LIN {X 0,Y 442.368,Z 762.06,A -85,B 0,C 180,E1 14751.098,E2 14751.098} C_VEL
LIN {X 0,Y 442.765,Z 762.06,A -85,B 0,C 180,E1 14758.998,E2 14758.998} C_VEL
LIN {X 0,Y 442.299,Z 762.06,A -85,B 0,C 180,E1 14768.863,E2 14768.863} C_VEL
LIN {X 0,Y 442.48,Z 764.15,A -85,B 0,C 180,E1 14772.989,E2 14772.989} C_VEL
LIN {X 0,Y 454.575,Z 779.497,A -85,B 0,C 180,E1 14779.866,E2 14779.866} C_VEL
LIN {X 0,Y 479.649,Z 812.394,A -85,B 0,C 180,E1 14788.603,E2 14788.603} C_VEL
LIN {X 0,Y 507.848,Z 858.532,A -85,B 0,C 180,E1 14795.89,E2 14795.89} C_VEL
LIN {X 0,Y 520.957,Z 891.034,A -85,B 0,C 180,E1 14799.521,E2 14799.521} C_VEL
LIN {X 0,Y 506.276,Z 963.742,A -85,B 0,C 180,E1 14802.79,E2 14802.79} C_VEL
LIN {X 0,Y 487.966,Z 1029.094,A -85,B 0,C 180,E1 14807.79,E2 14807.79} C_VEL
LIN {X 0,Y 469.666,Z 1084.518,A -85,B 0,C 180,E1 14814.467,E2 14814.467} C_VEL
LIN {X 0,Y 454.767,Z 1129.328,A -85,B 0,C 180,E1 14822.874,E2 14822.874} C_VEL
LIN {X 0,Y 446.413,Z 1161.096,A -85,B 0,C 180,E1 14832.529,E2 14832.529} C_VEL
LIN {X 0,Y 443.437,Z 1178.275,A -85,B 0,C 180,E1 14842.403,E2 14842.403} C_VEL
LIN {X 0,Y 443.471,Z 1182.026,A -85,B 0,C 180,E1 14850.982,E2 14850.982} C_VEL
LIN {X 0,Y 443.626,Z 1175.498,A -85,B 0,C 180,E1 14859.843,E2 14859.843} C_VEL
LIN {X 0,Y 447.223,Z 1156.157,A -85,B 0,C 180,E1 14869.308,E2 14869.308} C_VEL
LIN {X 0,Y 457.262,Z 1121.757,A -85,B 0,C 180,E1 14878.746,E2 14878.746} C_VEL
LIN {X 0,Y 473.14,Z 1074.147,A -85,B 0,C 180,E1 14886.926,E2 14886.926} C_VEL
LIN {X 0,Y 491.971,Z 1015.812,A -85,B 0,C 180,E1 14893.329,E2 14893.329} C_VEL
LIN {X 0,Y 509.871,Z 949.056,A -85,B 0,C 180,E1 14897.908,E2 14897.908} C_VEL
LIN {X 0,Y 520.404,Z 886.291,A -85,B 0,C 180,E1 14900.698,E2 14900.698} C_VEL
LIN {X 0,Y 494.713,Z 835.568,A -85,B 0,C 180,E1 14907.281,E2 14907.281} C_VEL
LIN {X 0,Y 467.97,Z 797.024,A -85,B 0,C 180,E1 14914.818,E2 14914.818} C_VEL
LIN {X 0,Y 451.114,Z 775.579,A -85,B 0,C 180,E1 14921.571,E2 14921.571} C_VEL
LIN {X 0,Y 445.46,Z 768.317,A -85,B 0,C 180,E1 14924.718,E2 14924.718} C_VEL
LIN {X 0,Y 442.777,Z 762.06,A -85,B 0,C 180,E1 14927.464,E2 14927.464} C_VEL
LIN {X 0,Y 442.754,Z 762.06,A -85,B 0,C 180,E1 14939.038,E2 14939.038} C_VEL
LIN {X 0,Y 442.287,Z 762.234,A -85,B 0,C 180,E1 14949.091,E2 14949.091} C_VEL
LIN {X 0,Y 459.966,Z 786.242,A -85,B 0,C 180,E1 14958.467,E2 14958.467} C_VEL
LIN {X 0,Y 486.214,Z 823.053,A -85,B 0,C 180,E1 14966.809,E2 14966.809} C_VEL
LIN {X 0,Y 512.137,Z 870.616,A -85,B 0,C 180,E1 14973.588,E2 14973.588} C_VEL
LIN {X 0,Y 521.201,Z 897.2,A -85,B 0,C 180,E1 14976.35,E2 14976.35} C_VEL
LIN {X 0,Y 506.051,Z 970.977,A -85,B 0,C 180,E1 14979.792,E2 14979.792} C_VEL
LIN {X 0,Y 487.203,Z 1040.281,A -85,B 0,C 180,E1 14985.118,E2 14985.118} C_VEL
LIN {X 0,Y 469.206,Z 1099.476,A -85,B 0,C 180,E1 14992.154,E2 14992.154} C_VEL
LIN {X 0,Y 454.918,Z 1147.637,A -85,B 0,C 180,E1 15000.758,E2 15000.758} C_VEL
LIN {X 0,Y 446.328,Z 1183.36,A -85,B 0,C 180,E1 15010.651,E2 15010.651} C_VEL
LIN {X 0,Y 443.387,Z 1202.811,A -85,B 0,C 180,E1 15020.151,E2 15020.151} C_VEL
LIN {X 0,Y 443.483,Z 1209.43,A -85,B 0,C 180,E1 15029.018,E2 15029.018} C_VEL
LIN {X 0,Y 443.218,Z 1205.935,A -85,B 0,C 180,E1 15037.185,E2 15037.185} C_VEL
LIN {X 0,Y 435.795,Z 1200.131,A -85,B 0,C 180,E1 15041.665,E2 15041.665} C_VEL
LIN {X 0,Y 439.135,Z 1178.691,A -85,B 0,C 180,E1 15051.258,E2 15051.258} C_VEL
LIN {X 0,Y 448.542,Z 1142.903,A -85,B 0,C 180,E1 15060.768,E2 15060.768} C_VEL
LIN {X 0,Y 464.675,Z 1092.053,A -85,B 0,C 180,E1 15069.522,E2 15069.522} C_VEL
LIN {X 0,Y 484.149,Z 1030.715,A -85,B 0,C 180,E1 15076.437,E2 15076.437} C_VEL
LIN {X 0,Y 503.041,Z 961.522,A -85,B 0,C 180,E1 15081.447,E2 15081.447} C_VEL
LIN {X 0,Y 515.029,Z 895.109,A -85,B 0,C 180,E1 15084.667,E2 15084.667} C_VEL
LIN {X 0,Y 495.626,Z 850.198,A -85,B 0,C 180,E1 15090.229,E2 15090.229} C_VEL
LIN {X 0,Y 470.178,Z 810.416,A -85,B 0,C 180,E1 15097.544,E2 15097.544} C_VEL
LIN {X 0,Y 450.662,Z 784.146,A -85,B 0,C 180,E1 15105.199,E2 15105.199} C_VEL
LIN {X 0,Y 439.348,Z 769.457,A -85,B 0,C 180,E1 15112.536,E2 15112.536} C_VEL
LIN {X 0,Y 434.707,Z 762.06,A -85,B 0,C 180,E1 15122.982,E2 15122.982} C_VEL
LIN {X 0,Y 441.317,Z 772.452,A -85,B 0,C 180,E1 15132.897,E2 15132.897} C_VEL
LIN {X 0,Y 453.083,Z 787.477,A -85,B 0,C 180,E1 15139.679,E2 15139.679} C_VEL
LIN {X 0,Y 477.143,Z 819.306,A -85,B 0,C 180,E1 15148.224,E2 15148.224} C_VEL
LIN {X 0,Y 504.175,Z 865.258,A -85,B 0,C 180,E1 15155.593,E2 15155.593} C_VEL
LIN {X 0,Y 515.619,Z 894.13,A -85,B 0,C 180,E1 15158.916,E2 15158.916} C_VEL
LIN {X 0,Y 500.351,Z 966.093,A -85,B 0,C 180,E1 15162.23,E2 15162.23} C_VEL
LIN {X 0,Y 481.899,Z 1029.755,A -85,B 0,C 180,E1 15167.17,E2 15167.17} C_VEL
LIN {X 0,Y 462.753,Z 1085.502,A -85,B 0,C 180,E1 15173.975,E2 15173.975} C_VEL
LIN {X 0,Y 447.354,Z 1129.813,A -85,B 0,C 180,E1 15182.435,E2 15182.435} C_VEL
LIN {X 0,Y 438.486,Z 1161.959,A -85,B 0,C 180,E1 15192.44,E2 15192.44} C_VEL
LIN {X 0,Y 435.483,Z 1178.22,A -85,B 0,C 180,E1 15201.995,E2 15201.995} C_VEL
LIN {X 0,Y 435.467,Z 1182.274,A -85,B 0,C 180,E1 15211,E2 15211} C_VEL
LIN {X 0,Y 435.666,Z 1175.758,A -85,B 0,C 180,E1 15220.025,E2 15220.025} C_VEL
LIN {X 0,Y 439.526,Z 1156.436,A -85,B 0,C 180,E1 15229.66,E2 15229.66} C_VEL
LIN {X 0,Y 450.076,Z 1122.065,A -85,B 0,C 180,E1 15239.249,E2 15239.249} C_VEL
LIN {X 0,Y 466.02,Z 1076.108,A -85,B 0,C 180,E1 15247.31,E2 15247.31} C_VEL
LIN {X 0,Y 485.667,Z 1017.605,A -85,B 0,C 180,E1 15253.862,E2 15253.862} C_VEL
LIN {X 0,Y 504.22,Z 950.876,A -85,B 0,C 180,E1 15258.515,E2 15258.515} C_VEL
LIN {X 0,Y 514.947,Z 889.714,A -85,B 0,C 180,E1 15261.319,E2 15261.319} C_VEL
LIN {X 0,Y 490.264,Z 840.18,A -85,B 0,C 180,E1 15267.986,E2 15267.986} C_VEL
LIN {X 0,Y 465.205,Z 803.405,A -85,B 0,C 180,E1 15275.378,E2 15275.378} C_VEL
LIN {X 0,Y 445.792,Z 777.155,A -85,B 0,C 180,E1 15283.961,E2 15283.961} C_VEL
LIN {X 0,Y 438.744,Z 769.012,A -85,B 0,C 180,E1 15289.052,E2 15289.052} C_VEL
LIN {X 0,Y 435.041,Z 762.06,A -85,B 0,C 180,E1 15297.037,E2 15297.037} C_VEL
LIN {X 0,Y 435.651,Z 765.907,A -85,B 0,C 180,E1 15303.516,E2 15303.516} C_VEL
LIN {X 0,Y 441.456,Z 772.745,A -85,B 0,C 180,E1 15309.42,E2 15309.42} C_VEL
LIN {X 0,Y 452.614,Z 786.488,A -85,B 0,C 180,E1 15315.806,E2 15315.806} C_VEL
LIN {X 0,Y 476.457,Z 819.233,A -85,B 0,C 180,E1 15324.436,E2 15324.436} C_VEL
LIN {X 0,Y 502.562,Z 864.703,A -85,B 0,C 180,E1 15331.736,E2 15331.736} C_VEL
LIN {X 0,Y 515.709,Z 900.205,A -85,B 0,C 180,E1 15335.759,E2 15335.759} C_VEL
LIN {X 0,Y 500.102,Z 973.092,A -85,B 0,C 180,E1 15339.231,E2 15339.231} C_VEL
LIN {X 0,Y 480.72,Z 1041.669,A -85,B 0,C 180,E1 15344.594,E2 15344.594} C_VEL
LIN {X 0,Y 461.544,Z 1102.125,A -85,B 0,C 180,E1 15351.963,E2 15351.963} C_VEL
LIN {X 0,Y 446.861,Z 1149.761,A -85,B 0,C 180,E1 15360.799,E2 15360.799} C_VEL
LIN {X 0,Y 438.175,Z 1184.384,A -85,B 0,C 180,E1 15370.802,E2 15370.802} C_VEL
LIN {X 0,Y 435.405,Z 1202.538,A -85,B 0,C 180,E1 15379.969,E2 15379.969} C_VEL
LIN {X 0,Y 435.475,Z 1209.182,A -85,B 0,C 180,E1 15389,E2 15389} C_VEL
LIN {X 0,Y 435.237,Z 1205.05,A -85,B 0,C 180,E1 15398.01,E2 15398.01} C_VEL
LIN {X 0,Y 435.795,Z 1200.131,A -85,B 0,C 180,E1 15401.665,E2 15401.665} C_VEL
LIN {X 0,Y 428.806,Z 1192.088,A -85,B 0,C 180,E1 15406.16,E2 15406.16} C_VEL
LIN {X 0,Y 436.129,Z 1161.529,A -85,B 0,C 180,E1 15416.713,E2 15416.713} C_VEL
LIN {X 0,Y 449.719,Z 1117.392,A -85,B 0,C 180,E1 15426.163,E2 15426.163} C_VEL
LIN {X 0,Y 468.68,Z 1060.673,A -85,B 0,C 180,E1 15434.079,E2 15434.079} C_VEL
LIN {X 0,Y 488.865,Z 994.656,A -85,B 0,C 180,E1 15440.057,E2 15440.057} C_VEL
LIN {X 0,Y 506.813,Z 921.365,A -85,B 0,C 180,E1 15444.141,E2 15444.141} C_VEL
LIN {X 0,Y 509.817,Z 899.368,A -85,B 0,C 180,E1 15445.171,E2 15445.171} C_VEL
LIN {X 0,Y 491.044,Z 854.603,A -85,B 0,C 180,E1 15450.91,E2 15450.91} C_VEL
LIN {X 0,Y 466.3,Z 815.129,A -85,B 0,C 180,E1 15458.437,E2 15458.437} C_VEL
LIN {X 0,Y 448.3,Z 791.119,A -85,B 0,C 180,E1 15465.833,E2 15465.833} C_VEL
LIN {X 0,Y 437.809,Z 777.136,A -85,B 0,C 180,E1 15473.01,E2 15473.01} C_VEL
LIN {X 0,Y 433.571,Z 769.978,A -85,B 0,C 180,E1 15482.989,E2 15482.989} C_VEL
LIN {X 0,Y 440.171,Z 780.615,A -85,B 0,C 180,E1 15492.804,E2 15492.804} C_VEL
LIN {X 0,Y 451.849,Z 795.781,A -85,B 0,C 180,E1 15499.607,E2 15499.607} C_VEL
LIN {X 0,Y 475.04,Z 827.197,A -85,B 0,C 180,E1 15508.017,E2 15508.017} C_VEL
LIN {X 0,Y 500.649,Z 872.118,A -85,B 0,C 180,E1 15515.323,E2 15515.323} C_VEL
LIN {X 0,Y 510.129,Z 897.959,A -85,B 0,C 180,E1 15518.334,E2 15518.334} C_VEL
LIN {X 0,Y 494.117,Z 969.785,A -85,B 0,C 180,E1 15521.742,E2 15521.742} C_VEL
LIN {X 0,Y 474.45,Z 1034.518,A -85,B 0,C 180,E1 15526.94,E2 15526.94} C_VEL
LIN {X 0,Y 454.998,Z 1088.953,A -85,B 0,C 180,E1 15533.856,E2 15533.856} C_VEL
LIN {X 0,Y 439.35,Z 1132.435,A -85,B 0,C 180,E1 15542.507,E2 15542.507} C_VEL
LIN {X 0,Y 430.405,Z 1163.295,A -85,B 0,C 180,E1 15552.575,E2 15552.575} C_VEL
LIN {X 0,Y 427.405,Z 1179.456,A -85,B 0,C 180,E1 15562.868,E2 15562.868} C_VEL
LIN {X 0,Y 427.468,Z 1182.521,A -85,B 0,C 180,E1 15571.018,E2 15571.018} C_VEL
LIN {X 0,Y 427.722,Z 1176.017,A -85,B 0,C 180,E1 15580.213,E2 15580.213} C_VEL
LIN {X 0,Y 431.848,Z 1156.711,A -85,B 0,C 180,E1 15590.025,E2 15590.025} C_VEL
LIN {X 0,Y 442.893,Z 1122.372,A -85,B 0,C 180,E1 15599.771,E2 15599.771} C_VEL
LIN {X 0,Y 459.545,Z 1076.449,A -85,B 0,C 180,E1 15607.927,E2 15607.927} C_VEL
LIN {X 0,Y 479.778,Z 1018.251,A -85,B 0,C 180,E1 15614.512,E2 15614.512} C_VEL
LIN {X 0,Y 498.685,Z 952.431,A -85,B 0,C 180,E1 15619.151,E2 15619.151} C_VEL
LIN {X 0,Y 509.807,Z 893.867,A -85,B 0,C 180,E1 15621.869,E2 15621.869} C_VEL
LIN {X 0,Y 486.092,Z 845.158,A -85,B 0,C 180,E1 15628.618,E2 15628.618} C_VEL
LIN {X 0,Y 460.424,Z 806.421,A -85,B 0,C 180,E1 15636.719,E2 15636.719} C_VEL
LIN {X 0,Y 443.003,Z 783.918,A -85,B 0,C 180,E1 15645.004,E2 15645.004} C_VEL
LIN {X 0,Y 437.511,Z 776.837,A -85,B 0,C 180,E1 15649.274,E2 15649.274} C_VEL
LIN {X 0,Y 433.267,Z 769.861,A -85,B 0,C 180,E1 15657.032,E2 15657.032} C_VEL
LIN {X 0,Y 435.072,Z 774.491,A -85,B 0,C 180,E1 15664.147,E2 15664.147} C_VEL
LIN {X 0,Y 440.298,Z 780.85,A -85,B 0,C 180,E1 15669.335,E2 15669.335} C_VEL
LIN {X 0,Y 451.153,Z 794.565,A -85,B 0,C 180,E1 15675.647,E2 15675.647} C_VEL
LIN {X 0,Y 473.701,Z 825.976,A -85,B 0,C 180,E1 15684.033,E2 15684.033} C_VEL
LIN {X 0,Y 498.655,Z 870.927,A -85,B 0,C 180,E1 15691.373,E2 15691.373} C_VEL
LIN {X 0,Y 510.181,Z 903.653,A -85,B 0,C 180,E1 15695.168,E2 15695.168} C_VEL
LIN {X 0,Y 494.109,Z 975.539,A -85,B 0,C 180,E1 15698.677,E2 15698.677} C_VEL
LIN {X 0,Y 474.019,Z 1043.819,A -85,B 0,C 180,E1 15704.127,E2 15704.127} C_VEL
LIN {X 0,Y 454.359,Z 1103.42,A -85,B 0,C 180,E1 15711.561,E2 15711.561} C_VEL
LIN {X 0,Y 439.179,Z 1150.529,A -85,B 0,C 180,E1 15720.522,E2 15720.522} C_VEL
LIN {X 0,Y 430.402,Z 1184.012,A -85,B 0,C 180,E1 15730.442,E2 15730.442} C_VEL
LIN {X 0,Y 427.424,Z 1202.261,A -85,B 0,C 180,E1 15739.78,E2 15739.78} C_VEL
LIN {X 0,Y 427.486,Z 1208.935,A -85,B 0,C 180,E1 15748.982,E2 15748.982} C_VEL
LIN {X 0,Y 427.272,Z 1204.781,A -85,B 0,C 180,E1 15758.16,E2 15758.16} C_VEL
LIN {X 0,Y 428.806,Z 1192.088,A -85,B 0,C 180,E1 15766.16,E2 15766.16} C_VEL
LIN {X 0,Y 422.844,Z 1181.735,A -85,B 0,C 180,E1 15770.681,E2 15770.681} C_VEL
LIN {X 0,Y 432.377,Z 1147.662,A -85,B 0,C 180,E1 15780.639,E2 15780.639} C_VEL
LIN {X 0,Y 448.741,Z 1099.846,A -85,B 0,C 180,E1 15789.621,E2 15789.621} C_VEL
LIN {X 0,Y 469.275,Z 1040.588,A -85,B 0,C 180,E1 15796.884,E2 15796.884} C_VEL
LIN {X 0,Y 489.459,Z 973.355,A -85,B 0,C 180,E1 15802.19,E2 15802.19} C_VEL
LIN {X 0,Y 504.46,Z 902.941,A -85,B 0,C 180,E1 15805.759,E2 15805.759} C_VEL
LIN {X 0,Y 486.135,Z 858.446,A -85,B 0,C 180,E1 15811.673,E2 15811.673} C_VEL
LIN {X 0,Y 462.362,Z 819.805,A -85,B 0,C 180,E1 15819.373,E2 15819.373} C_VEL
LIN {X 0,Y 442.895,Z 792.669,A -85,B 0,C 180,E1 15828.372,E2 15828.372} C_VEL
LIN {X 0,Y 435.286,Z 784.009,A -85,B 0,C 180,E1 15834.556,E2 15834.556} C_VEL
LIN {X 0,Y 432.597,Z 777.918,A -85,B 0,C 180,E1 15842.996,E2 15842.996} C_VEL
LIN {X 0,Y 439.113,Z 788.811,A -85,B 0,C 180,E1 15852.772,E2 15852.772} C_VEL
LIN {X 0,Y 451.323,Z 804.899,A -85,B 0,C 180,E1 15859.855,E2 15859.855} C_VEL
LIN {X 0,Y 474.1,Z 836.679,A -85,B 0,C 180,E1 15868.157,E2 15868.157} C_VEL
LIN {X 0,Y 498.176,Z 881.884,A -85,B 0,C 180,E1 15875.443,E2 15875.443} C_VEL
LIN {X 0,Y 504.581,Z 902.317,A -85,B 0,C 180,E1 15877.757,E2 15877.757} C_VEL
LIN {X 0,Y 487.858,Z 973.643,A -85,B 0,C 180,E1 15881.25,E2 15881.25} C_VEL
LIN {X 0,Y 467.667,Z 1037.478,A -85,B 0,C 180,E1 15886.526,E2 15886.526} C_VEL
LIN {X 0,Y 447.469,Z 1091.741,A -85,B 0,C 180,E1 15893.626,E2 15893.626} C_VEL
LIN {X 0,Y 431.699,Z 1133.776,A -85,B 0,C 180,E1 15902.262,E2 15902.262} C_VEL
LIN {X 0,Y 422.639,Z 1163.559,A -85,B 0,C 180,E1 15912.244,E2 15912.244} C_VEL
LIN {X 0,Y 419.42,Z 1179.707,A -85,B 0,C 180,E1 15922.732,E2 15922.732} C_VEL
LIN {X 0,Y 419.463,Z 1182.768,A -85,B 0,C 180,E1 15931.038,E2 15931.038} C_VEL
LIN {X 0,Y 419.777,Z 1176.274,A -85,B 0,C 180,E1 15940.409,E2 15940.409} C_VEL
LIN {X 0,Y 424.186,Z 1156.984,A -85,B 0,C 180,E1 15950.402,E2 15950.402} C_VEL
LIN {X 0,Y 435.766,Z 1122.674,A -85,B 0,C 180,E1 15960.308,E2 15960.308} C_VEL
LIN {X 0,Y 453.115,Z 1076.788,A -85,B 0,C 180,E1 15968.564,E2 15968.564} C_VEL
LIN {X 0,Y 474.033,Z 1018.657,A -85,B 0,C 180,E1 15975.199,E2 15975.199} C_VEL
LIN {X 0,Y 493.774,Z 951.807,A -85,B 0,C 180,E1 15979.922,E2 15979.922} C_VEL
LIN {X 0,Y 504.513,Z 897.743,A -85,B 0,C 180,E1 15982.444,E2 15982.444} C_VEL
LIN {X 0,Y 481.644,Z 849.459,A -85,B 0,C 180,E1 15989.365,E2 15989.365} C_VEL
LIN {X 0,Y 457.504,Z 812.799,A -85,B 0,C 180,E1 15997.4,E2 15997.4} C_VEL
LIN {X 0,Y 441.469,Z 791.511,A -85,B 0,C 180,E1 16005.333,E2 16005.333} C_VEL
LIN {X 0,Y 436.023,Z 784.509,A -85,B 0,C 180,E1 16009.744,E2 16009.744} C_VEL
LIN {X 0,Y 432.293,Z 777.802,A -85,B 0,C 180,E1 16017.03,E2 16017.03} C_VEL
LIN {X 0,Y 434.842,Z 783.442,A -85,B 0,C 180,E1 16025.154,E2 16025.154} C_VEL
LIN {X 0,Y 439.658,Z 789.715,A -85,B 0,C 180,E1 16029.647,E2 16029.647} C_VEL
LIN {X 0,Y 450.109,Z 803.222,A -85,B 0,C 180,E1 16035.685,E2 16035.685} C_VEL
LIN {X 0,Y 471.594,Z 833.871,A -85,B 0,C 180,E1 16043.833,E2 16043.833} C_VEL
LIN {X 0,Y 494.794,Z 877.553,A -85,B 0,C 180,E1 16051.064,E2 16051.064} C_VEL
LIN {X 0,Y 504.541,Z 907.941,A -85,B 0,C 180,E1 16054.593,E2 16054.593} C_VEL
LIN {X 0,Y 488.003,Z 978.599,A -85,B 0,C 180,E1 16058.148,E2 16058.148} C_VEL
LIN {X 0,Y 466.978,Z 1047.213,A -85,B 0,C 180,E1 16063.776,E2 16063.776} C_VEL
LIN {X 0,Y 446.76,Z 1106.04,A -85,B 0,C 180,E1 16071.35,E2 16071.35} C_VEL
LIN {X 0,Y 430.84,Z 1153.509,A -85,B 0,C 180,E1 16080.763,E2 16080.763} C_VEL
LIN {X 0,Y 421.937,Z 1186.372,A -85,B 0,C 180,E1 16091.125,E2 16091.125} C_VEL
LIN {X 0,Y 419.363,Z 1203.25,A -85,B 0,C 180,E1 16100.633,E2 16100.633} C_VEL
LIN {X 0,Y 419.477,Z 1208.687,A -85,B 0,C 180,E1 16108.962,E2 16108.962} C_VEL
LIN {X 0,Y 419.29,Z 1204.511,A -85,B 0,C 180,E1 16118.316,E2 16118.316} C_VEL
LIN {X 0,Y 421.958,Z 1187.595,A -85,B 0,C 180,E1 16128.327,E2 16128.327} C_VEL
LIN {X 0,Y 422.844,Z 1181.735,A -85,B 0,C 180,E1 16130.681,E2 16130.681} C_VEL
LIN {X 0,Y 418.248,Z 1169.611,A -85,B 0,C 180,E1 16135.187,E2 16135.187} C_VEL
LIN {X 0,Y 431.614,Z 1129.102,A -85,B 0,C 180,E1 16145.164,E2 16145.164} C_VEL
LIN {X 0,Y 450.871,Z 1076.056,A -85,B 0,C 180,E1 16153.605,E2 16153.605} C_VEL
LIN {X 0,Y 472.769,Z 1012.28,A -85,B 0,C 180,E1 16160.145,E2 16160.145} C_VEL
LIN {X 0,Y 492.26,Z 942.85,A -85,B 0,C 180,E1 16164.616,E2 16164.616} C_VEL
LIN {X 0,Y 499.077,Z 906.354,A -85,B 0,C 180,E1 16166.384,E2 16166.384} C_VEL
LIN {X 0,Y 481.278,Z 862.408,A -85,B 0,C 180,E1 16172.449,E2 16172.449} C_VEL
LIN {X 0,Y 459.047,Z 825.703,A -85,B 0,C 180,E1 16180.098,E2 16180.098} C_VEL
LIN {X 0,Y 441.194,Z 800.26,A -85,B 0,C 180,E1 16188.775,E2 16188.775} C_VEL
LIN {X 0,Y 433.745,Z 791.35,A -85,B 0,C 180,E1 16195.237,E2 16195.237} C_VEL
LIN {X 0,Y 431.624,Z 785.857,A -85,B 0,C 180,E1 16203.003,E2 16203.003} C_VEL
LIN {X 0,Y 437.985,Z 796.839,A -85,B 0,C 180,E1 16212.679,E2 16212.679} C_VEL
LIN {X 0,Y 452.325,Z 815.439,A -85,B 0,C 180,E1 16220.745,E2 16220.745} C_VEL
LIN {X 0,Y 475.731,Z 850.897,A -85,B 0,C 180,E1 16229.252,E2 16229.252} C_VEL
LIN {X 0,Y 497.417,Z 896.34,A -85,B 0,C 180,E1 16236.194,E2 16236.194} C_VEL
LIN {X 0,Y 498.983,Z 907.316,A -85,B 0,C 180,E1 16237.194,E2 16237.194} C_VEL
LIN {X 0,Y 481.662,Z 977.498,A -85,B 0,C 180,E1 16240.749,E2 16240.749} C_VEL
LIN {X 0,Y 460.518,Z 1041.371,A -85,B 0,C 180,E1 16246.192,E2 16246.192} C_VEL
LIN {X 0,Y 439.824,Z 1094.761,A -85,B 0,C 180,E1 16253.457,E2 16253.457} C_VEL
LIN {X 0,Y 423.715,Z 1135.961,A -85,B 0,C 180,E1 16262.274,E2 16262.274} C_VEL
LIN {X 0,Y 414.498,Z 1164.927,A -85,B 0,C 180,E1 16272.434,E2 16272.434} C_VEL
LIN {X 0,Y 411.441,Z 1179.957,A -85,B 0,C 180,E1 16282.59,E2 16282.59} C_VEL
LIN {X 0,Y 411.459,Z 1183.016,A -85,B 0,C 180,E1 16291.058,E2 16291.058} C_VEL
LIN {X 0,Y 411.824,Z 1176.532,A -85,B 0,C 180,E1 16300.612,E2 16300.612} C_VEL
LIN {X 0,Y 416.965,Z 1156.05,A -85,B 0,C 180,E1 16311.233,E2 16311.233} C_VEL
LIN {X 0,Y 429.339,Z 1121.155,A -85,B 0,C 180,E1 16321.27,E2 16321.27} C_VEL
LIN {X 0,Y 448.041,Z 1073.787,A -85,B 0,C 180,E1 16329.694,E2 16329.694} C_VEL
LIN {X 0,Y 469.613,Z 1015.141,A -85,B 0,C 180,E1 16336.27,E2 16336.27} C_VEL
LIN {X 0,Y 489.697,Z 948.44,A -85,B 0,C 180,E1 16340.856,E2 16340.856} C_VEL
LIN {X 0,Y 499.2,Z 901.472,A -85,B 0,C 180,E1 16343.052,E2 16343.052} C_VEL
LIN {X 0,Y 477.32,Z 854.135,A -85,B 0,C 180,E1 16350.098,E2 16350.098} C_VEL
LIN {X 0,Y 455.075,Z 819.55,A -85,B 0,C 180,E1 16357.919,E2 16357.919} C_VEL
LIN {X 0,Y 439.603,Z 798.612,A -85,B 0,C 180,E1 16365.907,E2 16365.907} C_VEL
LIN {X 0,Y 434.567,Z 792.146,A -85,B 0,C 180,E1 16370.217,E2 16370.217} C_VEL
LIN {X 0,Y 431.319,Z 785.742,A -85,B 0,C 180,E1 16377.027,E2 16377.027} C_VEL
LIN {X 0,Y 436.712,Z 793.622,A -85,B 0,C 180,E1 16387.949,E2 16387.949} C_VEL
LIN {X 0,Y 452.717,Z 816.474,A -85,B 0,C 180,E1 16397.347,E2 16397.347} C_VEL
LIN {X 0,Y 474.873,Z 851.14,A -85,B 0,C 180,E1 16405.52,E2 16405.52} C_VEL
LIN {X 0,Y 495.064,Z 894.701,A -85,B 0,C 180,E1 16412.168,E2 16412.168} C_VEL
LIN {X 0,Y 499.112,Z 911.594,A -85,B 0,C 180,E1 16413.987,E2 16413.987} C_VEL
LIN {X 0,Y 481.692,Z 982.576,A -85,B 0,C 180,E1 16417.665,E2 16417.665} C_VEL
LIN {X 0,Y 460.132,Z 1050.013,A -85,B 0,C 180,E1 16423.35,E2 16423.35} C_VEL
LIN {X 0,Y 439.235,Z 1108.191,A -85,B 0,C 180,E1 16431.065,E2 16431.065} C_VEL
LIN {X 0,Y 423.17,Z 1154.2,A -85,B 0,C 180,E1 16440.476,E2 16440.476} C_VEL
LIN {X 0,Y 414.162,Z 1186.073,A -85,B 0,C 180,E1 16450.756,E2 16450.756} C_VEL
LIN {X 0,Y 411.374,Z 1202.97,A -85,B 0,C 180,E1 16460.449,E2 16460.449} C_VEL
LIN {X 0,Y 411.47,Z 1208.439,A -85,B 0,C 180,E1 16468.942,E2 16468.942} C_VEL
LIN {X 0,Y 411.316,Z 1204.241,A -85,B 0,C 180,E1 16478.479,E2 16478.479} C_VEL
LIN {X 0,Y 414.116,Z 1187.293,A -85,B 0,C 180,E1 16488.687,E2 16488.687} C_VEL
LIN {X 0,Y 418.248,Z 1169.611,A -85,B 0,C 180,E1 16495.187,E2 16495.187} C_VEL
LIN {X 0,Y 415.04,Z 1155.527,A -85,B 0,C 180,E1 16499.67,E2 16499.67} C_VEL
LIN {X 0,Y 431.336,Z 1110.915,A -85,B 0,C 180,E1 16509.128,E2 16509.128} C_VEL
LIN {X 0,Y 453.186,Z 1053.242,A -85,B 0,C 180,E1 16517.016,E2 16517.016} C_VEL
LIN {X 0,Y 475.06,Z 987.25,A -85,B 0,C 180,E1 16522.799,E2 16522.799} C_VEL
LIN {X 0,Y 494.251,Z 911.935,A -85,B 0,C 180,E1 16526.791,E2 16526.791} C_VEL
LIN {X 0,Y 478.267,Z 869.924,A -85,B 0,C 180,E1 16532.645,E2 16532.645} C_VEL
LIN {X 0,Y 456.95,Z 833.052,A -85,B 0,C 180,E1 16540.39,E2 16540.39} C_VEL
LIN {X 0,Y 439.563,Z 807.774,A -85,B 0,C 180,E1 16549.158,E2 16549.158} C_VEL
LIN {X 0,Y 432.303,Z 798.658,A -85,B 0,C 180,E1 16555.879,E2 16555.879} C_VEL
LIN {X 0,Y 430.731,Z 793.915,A -85,B 0,C 180,E1 16563.515,E2 16563.515} C_VEL
LIN {X 0,Y 437.242,Z 805.417,A -85,B 0,C 180,E1 16572.892,E2 16572.892} C_VEL
LIN {X 0,Y 451.563,Z 824.899,A -85,B 0,C 180,E1 16580.964,E2 16580.964} C_VEL
LIN {X 0,Y 473.017,Z 858.348,A -85,B 0,C 180,E1 16589.012,E2 16589.012} C_VEL
LIN {X 0,Y 493.63,Z 904.302,A -85,B 0,C 180,E1 16596.1,E2 16596.1} C_VEL
LIN {X 0,Y 485.008,Z 947.709,A -85,B 0,C 180,E1 16598.226,E2 16598.226} C_VEL
LIN {X 0,Y 464.821,Z 1013.88,A -85,B 0,C 180,E1 16602.773,E2 16602.773} C_VEL
LIN {X 0,Y 442.201,Z 1072.822,A -85,B 0,C 180,E1 16609.327,E2 16609.327} C_VEL
LIN {X 0,Y 422.11,Z 1121.19,A -85,B 0,C 180,E1 16617.961,E2 16617.961} C_VEL
LIN {X 0,Y 409.445,Z 1155.059,A -85,B 0,C 180,E1 16627.767,E2 16627.767} C_VEL
LIN {X 0,Y 404.174,Z 1175.424,A -85,B 0,C 180,E1 16638.093,E2 16638.093} C_VEL
LIN {X 0,Y 403.13,Z 1182.817,A -85,B 0,C 180,E1 16646.767,E2 16646.767} C_VEL
LIN {X 0,Y 403.276,Z 1181.773,A -85,B 0,C 180,E1 16655.397,E2 16655.397} C_VEL
LIN {X 0,Y 405.333,Z 1170.222,A -85,B 0,C 180,E1 16665.185,E2 16665.185} C_VEL
LIN {X 0,Y 412.688,Z 1145.441,A -85,B 0,C 180,E1 16675.458,E2 16675.458} C_VEL
LIN {X 0,Y 428.364,Z 1106.05,A -85,B 0,C 180,E1 16685.122,E2 16685.122} C_VEL
LIN {X 0,Y 449.917,Z 1053.779,A -85,B 0,C 180,E1 16693.046,E2 16693.046} C_VEL
LIN {X 0,Y 472.053,Z 991.825,A -85,B 0,C 180,E1 16698.909,E2 16698.909} C_VEL
LIN {X 0,Y 491.121,Z 921.335,A -85,B 0,C 180,E1 16702.936,E2 16702.936} C_VEL
LIN {X 0,Y 493.496,Z 903.941,A -85,B 0,C 180,E1 16703.836,E2 16703.836} C_VEL
LIN {X 0,Y 472.023,Z 856.912,A -85,B 0,C 180,E1 16711.184,E2 16711.184} C_VEL
LIN {X 0,Y 449.787,Z 821.777,A -85,B 0,C 180,E1 16719.708,E2 16719.708} C_VEL
LIN {X 0,Y 434.933,Z 800.853,A -85,B 0,C 180,E1 16728.955,E2 16728.955} C_VEL
LIN {X 0,Y 430.345,Z 793.682,A -85,B 0,C 180,E1 16737.025,E2 16737.025} C_VEL
LIN {X 0,Y 435.542,Z 801.809,A -85,B 0,C 180,E1 16747.844,E2 16747.844} C_VEL
LIN {X 0,Y 450.871,Z 824.07,A -85,B 0,C 180,E1 16757.105,E2 16757.105} C_VEL
LIN {X 0,Y 471.938,Z 858.335,A -85,B 0,C 180,E1 16765.243,E2 16765.243} C_VEL
LIN {X 0,Y 490.999,Z 901.736,A -85,B 0,C 180,E1 16771.964,E2 16771.964} C_VEL
LIN {X 0,Y 493.539,Z 915.76,A -85,B 0,C 180,E1 16773.404,E2 16773.404} C_VEL
LIN {X 0,Y 475.942,Z 984.617,A -85,B 0,C 180,E1 16777.041,E2 16777.041} C_VEL
LIN {X 0,Y 453.589,Z 1051.837,A -85,B 0,C 180,E1 16782.821,E2 16782.821} C_VEL
LIN {X 0,Y 432.318,Z 1108.782,A -85,B 0,C 180,E1 16790.522,E2 16790.522} C_VEL
LIN {X 0,Y 415.713,Z 1154.354,A -85,B 0,C 180,E1 16800.031,E2 16800.031} C_VEL
LIN {X 0,Y 406.036,Z 1186.983,A -85,B 0,C 180,E1 16810.923,E2 16810.923} C_VEL
LIN {X 0,Y 403.416,Z 1202.702,A -85,B 0,C 180,E1 16820.259,E2 16820.259} C_VEL
LIN {X 0,Y 403.461,Z 1208.191,A -85,B 0,C 180,E1 16828.921,E2 16828.921} C_VEL
LIN {X 0,Y 403.336,Z 1203.974,A -85,B 0,C 180,E1 16838.648,E2 16838.648} C_VEL
LIN {X 0,Y 406.265,Z 1187.004,A -85,B 0,C 180,E1 16849.062,E2 16849.062} C_VEL
LIN {X 0,Y 415.04,Z 1155.527,A -85,B 0,C 180,E1 16859.67,E2 16859.67} C_VEL
LIN {X 0,Y 413.408,Z 1139.818,A -85,B 0,C 180,E1 16864.07,E2 16864.07} C_VEL
LIN {X 0,Y 433.49,Z 1088.836,A -85,B 0,C 180,E1 16873.272,E2 16873.272} C_VEL
LIN {X 0,Y 456.696,Z 1027.449,A -85,B 0,C 180,E1 16880.347,E2 16880.347} C_VEL
LIN {X 0,Y 478.25,Z 959.226,A -85,B 0,C 180,E1 16885.283,E2 16885.283} C_VEL
LIN {X 0,Y 488.388,Z 912.77,A -85,B 0,C 180,E1 16887.719,E2 16887.719} C_VEL
LIN {X 0,Y 471.557,Z 869.997,A -85,B 0,C 180,E1 16894.135,E2 16894.135} C_VEL
LIN {X 0,Y 450.953,Z 834.395,A -85,B 0,C 180,E1 16902.346,E2 16902.346} C_VEL
LIN {X 0,Y 436.635,Z 813.928,A -85,B 0,C 180,E1 16910.475,E2 16910.475} C_VEL
LIN {X 0,Y 430.162,Z 803.999,A -85,B 0,C 180,E1 16918.21,E2 16918.21} C_VEL
LIN {X 0,Y 429.85,Z 803.306,A -85,B 0,C 180,E1 16924.473,E2 16924.473} C_VEL
LIN {X 0,Y 436.045,Z 813.254,A -85,B 0,C 180,E1 16932.736,E2 16932.736} C_VEL
LIN {X 0,Y 450.036,Z 832.984,A -85,B 0,C 180,E1 16940.856,E2 16940.856} C_VEL
LIN {X 0,Y 469.853,Z 865.261,A -85,B 0,C 180,E1 16948.698,E2 16948.698} C_VEL
LIN {X 0,Y 489.117,Z 910.05,A -85,B 0,C 180,E1 16955.724,E2 16955.724} C_VEL
LIN {X 0,Y 470.71,Z 980.426,A -85,B 0,C 180,E1 16959.395,E2 16959.395} C_VEL
LIN {X 0,Y 448.149,Z 1043.854,A -85,B 0,C 180,E1 16964.953,E2 16964.953} C_VEL
LIN {X 0,Y 425.933,Z 1097.021,A -85,B 0,C 180,E1 16972.433,E2 16972.433} C_VEL
LIN {X 0,Y 408.317,Z 1138.643,A -85,B 0,C 180,E1 16981.813,E2 16981.813} C_VEL
LIN {X 0,Y 398.382,Z 1167.21,A -85,B 0,C 180,E1 16992.611,E2 16992.611} C_VEL
LIN {X 0,Y 395.52,Z 1180.456,A -85,B 0,C 180,E1 17002.29,E2 17002.29} C_VEL
LIN {X 0,Y 395.475,Z 1183.51,A -85,B 0,C 180,E1 17011.101,E2 17011.101} C_VEL
LIN {X 0,Y 395.942,Z 1177.044,A -85,B 0,C 180,E1 17021.043,E2 17021.043} C_VEL
LIN {X 0,Y 401.444,Z 1157.504,A -85,B 0,C 180,E1 17031.737,E2 17031.737} C_VEL
LIN {X 0,Y 415.047,Z 1122.354,A -85,B 0,C 180,E1 17042.316,E2 17042.316} C_VEL
LIN {X 0,Y 435.094,Z 1075.555,A -85,B 0,C 180,E1 17050.91,E2 17050.91} C_VEL
LIN {X 0,Y 458.192,Z 1016.857,A -85,B 0,C 180,E1 17057.654,E2 17057.654} C_VEL
LIN {X 0,Y 479.367,Z 950.83,A -85,B 0,C 180,E1 17062.271,E2 17062.271} C_VEL
LIN {X 0,Y 488.691,Z 908.835,A -85,B 0,C 180,E1 17064.323,E2 17064.323} C_VEL
LIN {X 0,Y 468.249,Z 862.746,A -85,B 0,C 180,E1 17071.723,E2 17071.723} C_VEL
LIN {X 0,Y 447.797,Z 829.159,A -85,B 0,C 180,E1 17080.046,E2 17080.046} C_VEL
LIN {X 0,Y 433.699,Z 808.66,A -85,B 0,C 180,E1 17089.179,E2 17089.179} C_VEL
LIN {X 0,Y 429.339,Z 801.641,A -85,B 0,C 180,E1 17099.008,E2 17099.008} C_VEL
LIN {X 0,Y 435.636,Z 812.715,A -85,B 0,C 180,E1 17108.915,E2 17108.915} C_VEL
LIN {X 0,Y 448.749,Z 831.194,A -85,B 0,C 180,E1 17116.729,E2 17116.729} C_VEL
LIN {X 0,Y 468.865,Z 865.475,A -85,B 0,C 180,E1 17124.972,E2 17124.972} C_VEL
LIN {X 0,Y 486.891,Z 908.647,A -85,B 0,C 180,E1 17131.74,E2 17131.74} C_VEL
LIN {X 0,Y 488.095,Z 919.228,A -85,B 0,C 180,E1 17132.773,E2 17132.773} C_VEL
LIN {X 0,Y 469.551,Z 988.705,A -85,B 0,C 180,E1 17136.561,E2 17136.561} C_VEL
LIN {X 0,Y 446.67,Z 1054.746,A -85,B 0,C 180,E1 17142.408,E2 17142.408} C_VEL
LIN {X 0,Y 424.402,Z 1111.794,A -85,B 0,C 180,E1 17150.381,E2 17150.381} C_VEL
LIN {X 0,Y 407.151,Z 1157.382,A -85,B 0,C 180,E1 17160.353,E2 17160.353} C_VEL
LIN {X 0,Y 397.892,Z 1187.898,A -85,B 0,C 180,E1 17171.095,E2 17171.095} C_VEL
LIN {X 0,Y 395.359,Z 1203.707,A -85,B 0,C 180,E1 17181.172,E2 17181.172} C_VEL
LIN {X 0,Y 395.059,Z 1207.932,A -85,B 0,C 180,E1 17191.098,E2 17191.098} C_VEL
LIN {X 0,Y 395.71,Z 1201.277,A -85,B 0,C 180,E1 17200.96,E2 17200.96} C_VEL
LIN {X 0,Y 399.366,Z 1181.535,A -85,B 0,C 180,E1 17211.669,E2 17211.669} C_VEL
LIN {X 0,Y 410.092,Z 1148.489,A -85,B 0,C 180,E1 17222.004,E2 17222.004} C_VEL
LIN {X 0,Y 413.408,Z 1139.818,A -85,B 0,C 180,E1 17224.07,E2 17224.07} C_VEL
LIN {X 0,Y 413.573,Z 1122.299,A -85,B 0,C 180,E1 17228.355,E2 17228.355} C_VEL
LIN {X 0,Y 435.874,Z 1067.812,A -85,B 0,C 180,E1 17236.818,E2 17236.818} C_VEL
LIN {X 0,Y 459.548,Z 1003.732,A -85,B 0,C 180,E1 17243.15,E2 17243.15} C_VEL
LIN {X 0,Y 480.974,Z 930.828,A -85,B 0,C 180,E1 17247.524,E2 17247.524} C_VEL
LIN {X 0,Y 482.912,Z 915.625,A -85,B 0,C 180,E1 17248.447,E2 17248.447} C_VEL
LIN {X 0,Y 466.763,Z 873.802,A -85,B 0,C 180,E1 17255.027,E2 17255.027} C_VEL
LIN {X 0,Y 447.522,Z 839.859,A -85,B 0,C 180,E1 17263.224,E2 17263.224} C_VEL
LIN {X 0,Y 433.831,Z 819.251,A -85,B 0,C 180,E1 17271.935,E2 17271.935} C_VEL
LIN {X 0,Y 428.657,Z 809.656,A -85,B 0,C 180,E1 17280.994,E2 17280.994} C_VEL
LIN {X 0,Y 433.908,Z 819.444,A -85,B 0,C 180,E1 17291.774,E2 17291.774} C_VEL
LIN {X 0,Y 447.974,Z 840.316,A -85,B 0,C 180,E1 17300.556,E2 17300.556} C_VEL
LIN {X 0,Y 466.842,Z 872.523,A -85,B 0,C 180,E1 17308.436,E2 17308.436} C_VEL
LIN {X 0,Y 483.831,Z 914.442,A -85,B 0,C 180,E1 17315.135,E2 17315.135} C_VEL
LIN {X 0,Y 464.644,Z 983.825,A -85,B 0,C 180,E1 17318.84,E2 17318.84} C_VEL
LIN {X 0,Y 441.277,Z 1046.911,A -85,B 0,C 180,E1 17324.515,E2 17324.515} C_VEL
LIN {X 0,Y 418.151,Z 1100.17,A -85,B 0,C 180,E1 17332.268,E2 17332.268} C_VEL
LIN {X 0,Y 400.415,Z 1140.574,A -85,B 0,C 180,E1 17341.746,E2 17341.746} C_VEL
LIN {X 0,Y 390.129,Z 1169.027,A -85,B 0,C 180,E1 17353.052,E2 17353.052} C_VEL
LIN {X 0,Y 387.547,Z 1180.705,A -85,B 0,C 180,E1 17362.13,E2 17362.13} C_VEL
LIN {X 0,Y 387.28,Z 1183.552,A -85,B 0,C 180,E1 17372.593,E2 17372.593} C_VEL
LIN {X 0,Y 388.37,Z 1175.798,A -85,B 0,C 180,E1 17382.404,E2 17382.404} C_VEL
LIN {X 0,Y 395.192,Z 1153.653,A -85,B 0,C 180,E1 17393.764,E2 17393.764} C_VEL
LIN {X 0,Y 410.07,Z 1117.998,A -85,B 0,C 180,E1 17404.018,E2 17404.018} C_VEL
LIN {X 0,Y 431.825,Z 1069.304,A -85,B 0,C 180,E1 17412.584,E2 17412.584} C_VEL
LIN {X 0,Y 455.371,Z 1010.442,A -85,B 0,C 180,E1 17419.014,E2 17419.014} C_VEL
LIN {X 0,Y 476.872,Z 942.438,A -85,B 0,C 180,E1 17423.514,E2 17423.514} C_VEL
LIN {X 0,Y 483.275,Z 912.058,A -85,B 0,C 180,E1 17425.051,E2 17425.051} C_VEL
LIN {X 0,Y 463.52,Z 866.471,A -85,B 0,C 180,E1 17432.67,E2 17432.67} C_VEL
LIN {X 0,Y 444.723,Z 835.227,A -85,B 0,C 180,E1 17440.916,E2 17440.916} C_VEL
LIN {X 0,Y 432.47,Z 816.481,A -85,B 0,C 180,E1 17449.403,E2 17449.403} C_VEL
LIN {X 0,Y 428.364,Z 809.582,A -85,B 0,C 180,E1 17459.006,E2 17459.006} C_VEL
LIN {X 0,Y 434.55,Z 820.853,A -85,B 0,C 180,E1 17468.937,E2 17468.937} C_VEL
LIN {X 0,Y 447.93,Z 840.789,A -85,B 0,C 180,E1 17477.077,E2 17477.077} C_VEL
LIN {X 0,Y 466.838,Z 874.646,A -85,B 0,C 180,E1 17485.089,E2 17485.089} C_VEL
LIN {X 0,Y 483.472,Z 918.455,A -85,B 0,C 180,E1 17491.91,E2 17491.91} C_VEL
LIN {X 0,Y 463.866,Z 990.631,A -85,B 0,C 180,E1 17495.911,E2 17495.911} C_VEL
LIN {X 0,Y 440.118,Z 1056.693,A -85,B 0,C 180,E1 17501.868,E2 17501.868} C_VEL
LIN {X 0,Y 416.711,Z 1114.349,A -85,B 0,C 180,E1 17510.155,E2 17510.155} C_VEL
LIN {X 0,Y 399.013,Z 1159.338,A -85,B 0,C 180,E1 17520.388,E2 17520.388} C_VEL
LIN {X 0,Y 389.786,Z 1188.819,A -85,B 0,C 180,E1 17531.276,E2 17531.276} C_VEL
LIN {X 0,Y 387.37,Z 1203.449,A -85,B 0,C 180,E1 17540.988,E2 17540.988} C_VEL
LIN {X 0,Y 387.062,Z 1207.685,A -85,B 0,C 180,E1 17551.12,E2 17551.12} C_VEL
LIN {X 0,Y 387.742,Z 1201.137,A -85,B 0,C 180,E1 17561.083,E2 17561.083} C_VEL
LIN {X 0,Y 391.337,Z 1182.507,A -85,B 0,C 180,E1 17571.599,E2 17571.599} C_VEL
LIN {X 0,Y 402.467,Z 1149.549,A -85,B 0,C 180,E1 17582.296,E2 17582.296} C_VEL
LIN {X 0,Y 413.573,Z 1122.299,A -85,B 0,C 180,E1 17588.355,E2 17588.355} C_VEL
LIN {X 0,Y 414.829,Z 1103.252,A -85,B 0,C 180,E1 17592.5,E2 17592.5} C_VEL
LIN {X 0,Y 439.328,Z 1044.555,A -85,B 0,C 180,E1 17600.246,E2 17600.246} C_VEL
LIN {X 0,Y 463.116,Z 977.722,A -85,B 0,C 180,E1 17605.771,E2 17605.771} C_VEL
LIN {X 0,Y 478.022,Z 920.595,A -85,B 0,C 180,E1 17608.916,E2 17608.916} C_VEL
LIN {X 0,Y 462.703,Z 879.268,A -85,B 0,C 180,E1 17615.599,E2 17615.599} C_VEL
LIN {X 0,Y 443.88,Z 844.404,A -85,B 0,C 180,E1 17624.294,E2 17624.294} C_VEL
LIN {X 0,Y 431.245,Z 824.553,A -85,B 0,C 180,E1 17633.411,E2 17633.411} C_VEL
LIN {X 0,Y 427.756,Z 817.744,A -85,B 0,C 180,E1 17643.285,E2 17643.285} C_VEL
LIN {X 0,Y 434.08,Z 829.79,A -85,B 0,C 180,E1 17652.977,E2 17652.977} C_VEL
LIN {X 0,Y 448.171,Z 851.328,A -85,B 0,C 180,E1 17661.445,E2 17661.445} C_VEL
LIN {X 0,Y 466.433,Z 885.744,A -85,B 0,C 180,E1 17669.324,E2 17669.324} C_VEL
LIN {X 0,Y 478.455,Z 918.6,A -85,B 0,C 180,E1 17674.501,E2 17674.501} C_VEL
LIN {X 0,Y 458.329,Z 988.172,A -85,B 0,C 180,E1 17678.345,E2 17678.345} C_VEL
LIN {X 0,Y 434.259,Z 1050.352,A -85,B 0,C 180,E1 17684.107,E2 17684.107} C_VEL
LIN {X 0,Y 411.004,Z 1101.894,A -85,B 0,C 180,E1 17691.83,E2 17691.83} C_VEL
LIN {X 0,Y 392.397,Z 1142.739,A -85,B 0,C 180,E1 17701.745,E2 17701.745} C_VEL
LIN {X 0,Y 382.339,Z 1169.286,A -85,B 0,C 180,E1 17712.696,E2 17712.696} C_VEL
LIN {X 0,Y 379.576,Z 1180.955,A -85,B 0,C 180,E1 17721.964,E2 17721.964} C_VEL
LIN {X 0,Y 379.474,Z 1184.004,A -85,B 0,C 180,E1 17731.147,E2 17731.147} C_VEL
LIN {X 0,Y 380.327,Z 1176.627,A -85,B 0,C 180,E1 17742.223,E2 17742.223} C_VEL
LIN {X 0,Y 387.252,Z 1155.083,A -85,B 0,C 180,E1 17753.8,E2 17753.8} C_VEL
LIN {X 0,Y 402.731,Z 1119.41,A -85,B 0,C 180,E1 17764.412,E2 17764.412} C_VEL
LIN {X 0,Y 424.937,Z 1071.56,A -85,B 0,C 180,E1 17773.048,E2 17773.048} C_VEL
LIN {X 0,Y 449.329,Z 1012.918,A -85,B 0,C 180,E1 17779.612,E2 17779.612} C_VEL
LIN {X 0,Y 471.602,Z 945.155,A -85,B 0,C 180,E1 17784.192,E2 17784.192} C_VEL
LIN {X 0,Y 477.98,Z 915.781,A -85,B 0,C 180,E1 17785.715,E2 17785.715} C_VEL
LIN {X 0,Y 459.585,Z 871.714,A -85,B 0,C 180,E1 17793.346,E2 17793.346} C_VEL
LIN {X 0,Y 441.747,Z 841.213,A -85,B 0,C 180,E1 17801.721,E2 17801.721} C_VEL
LIN {X 0,Y 430.955,Z 824.206,A -85,B 0,C 180,E1 17809.774,E2 17809.774} C_VEL
LIN {X 0,Y 427.388,Z 817.521,A -85,B 0,C 180,E1 17819.003,E2 17819.003} C_VEL
LIN {X 0,Y 433.291,Z 828.887,A -85,B 0,C 180,E1 17828.9,E2 17828.9} C_VEL
LIN {X 0,Y 446.874,Z 849.808,A -85,B 0,C 180,E1 17837.374,E2 17837.374} C_VEL
LIN {X 0,Y 465.227,Z 885.636,A -85,B 0,C 180,E1 17845.561,E2 17845.561} C_VEL
LIN {X 0,Y 478.158,Z 923.034,A -85,B 0,C 180,E1 17851.34,E2 17851.34} C_VEL
LIN {X 0,Y 458.332,Z 992.292,A -85,B 0,C 180,E1 17855.226,E2 17855.226} C_VEL
LIN {X 0,Y 433.364,Z 1059.318,A -85,B 0,C 180,E1 17861.393,E2 17861.393} C_VEL
LIN {X 0,Y 409.727,Z 1115.275,A -85,B 0,C 180,E1 17869.627,E2 17869.627} C_VEL
LIN {X 0,Y 391.372,Z 1160.049,A -85,B 0,C 180,E1 17880.071,E2 17880.071} C_VEL
LIN {X 0,Y 381.688,Z 1189.741,A -85,B 0,C 180,E1 17891.464,E2 17891.464} C_VEL
LIN {X 0,Y 379.349,Z 1204.143,A -85,B 0,C 180,E1 17901.955,E2 17901.955} C_VEL
LIN {X 0,Y 379.063,Z 1207.437,A -85,B 0,C 180,E1 17911.144,E2 17911.144} C_VEL
LIN {X 0,Y 379.794,Z 1200.553,A -85,B 0,C 180,E1 17921.615,E2 17921.615} C_VEL
LIN {X 0,Y 383.983,Z 1180.832,A -85,B 0,C 180,E1 17932.646,E2 17932.646} C_VEL
LIN {X 0,Y 395.929,Z 1147.661,A -85,B 0,C 180,E1 17943.357,E2 17943.357} C_VEL
LIN {X 0,Y 414.829,Z 1103.252,A -85,B 0,C 180,E1 17952.5,E2 17952.5} C_VEL
LIN {X 0,Y 417.817,Z 1082.444,A -85,B 0,C 180,E1 17956.441,E2 17956.441} C_VEL
LIN {X 0,Y 443.666,Z 1019.755,A -85,B 0,C 180,E1 17963.439,E2 17963.439} C_VEL
LIN {X 0,Y 466.505,Z 951.33,A -85,B 0,C 180,E1 17968.129,E2 17968.129} C_VEL
LIN {X 0,Y 472.865,Z 924.245,A -85,B 0,C 180,E1 17969.569,E2 17969.569} C_VEL
LIN {X 0,Y 458.034,Z 883.287,A -85,B 0,C 180,E1 17976.469,E2 17976.469} C_VEL
LIN {X 0,Y 440.749,Z 850.672,A -85,B 0,C 180,E1 17985.075,E2 17985.075} C_VEL
LIN {X 0,Y 429.841,Z 832.303,A -85,B 0,C 180,E1 17993.644,E2 17993.644} C_VEL
LIN {X 0,Y 426.595,Z 825.728,A -85,B 0,C 180,E1 18003.294,E2 18003.294} C_VEL
LIN {X 0,Y 434.303,Z 839.272,A -85,B 0,C 180,E1 18014.075,E2 18014.075} C_VEL
LIN {X 0,Y 450.743,Z 867.557,A -85,B 0,C 180,E1 18023.614,E2 18023.614} C_VEL
LIN {X 0,Y 467.127,Z 903.186,A -85,B 0,C 180,E1 18030.899,E2 18030.899} C_VEL
LIN {X 0,Y 472.971,Z 923.446,A -85,B 0,C 180,E1 18033.882,E2 18033.882} C_VEL
LIN {X 0,Y 452.38,Z 991.497,A -85,B 0,C 180,E1 18037.757,E2 18037.757} C_VEL
LIN {X 0,Y 427.504,Z 1053.235,A -85,B 0,C 180,E1 18043.619,E2 18043.619} C_VEL
LIN {X 0,Y 403.252,Z 1105.04,A -85,B 0,C 180,E1 18051.649,E2 18051.649} C_VEL
LIN {X 0,Y 384.38,Z 1144.766,A -85,B 0,C 180,E1 18061.745,E2 18061.745} C_VEL
LIN {X 0,Y 373.839,Z 1171.421,A -85,B 0,C 180,E1 18073.506,E2 18073.506} C_VEL
LIN {X 0,Y 371.399,Z 1182.824,A -85,B 0,C 180,E1 18084.143,E2 18084.143} C_VEL
LIN {X 0,Y 371.259,Z 1183.76,A -85,B 0,C 180,E1 18093.515,E2 18093.515} C_VEL
LIN {X 0,Y 373.039,Z 1174.809,A -85,B 0,C 180,E1 18104.12,E2 18104.12} C_VEL
LIN {X 0,Y 381.057,Z 1151.782,A -85,B 0,C 180,E1 18115.732,E2 18115.732} C_VEL
LIN {X 0,Y 398.127,Z 1114.996,A -85,B 0,C 180,E1 18126.189,E2 18126.189} C_VEL
LIN {X 0,Y 422.096,Z 1065.033,A -85,B 0,C 180,E1 18134.766,E2 18134.766} C_VEL
LIN {X 0,Y 447.536,Z 1004.235,A -85,B 0,C 180,E1 18141.165,E2 18141.165} C_VEL
LIN {X 0,Y 469.809,Z 935.01,A -85,B 0,C 180,E1 18145.517,E2 18145.517} C_VEL
LIN {X 0,Y 472.73,Z 919.563,A -85,B 0,C 180,E1 18146.391,E2 18146.391} C_VEL
LIN {X 0,Y 455.484,Z 876.771,A -85,B 0,C 180,E1 18154.086,E2 18154.086} C_VEL
LIN {X 0,Y 438.081,Z 845.43,A -85,B 0,C 180,E1 18163.023,E2 18163.023} C_VEL
LIN {X 0,Y 428.777,Z 831.453,A -85,B 0,C 180,E1 18170.855,E2 18170.855} C_VEL
LIN {X 0,Y 426.236,Z 825.437,A -85,B 0,C 180,E1 18179.001,E2 18179.001} C_VEL
LIN {X 0,Y 432.297,Z 837.218,A -85,B 0,C 180,E1 18189.111,E2 18189.111} C_VEL
LIN {X 0,Y 445.238,Z 858.63,A -85,B 0,C 180,E1 18197.504,E2 18197.504} C_VEL
LIN {X 0,Y 462.075,Z 893.251,A -85,B 0,C 180,E1 18205.404,E2 18205.404} C_VEL
LIN {X 0,Y 472.691,Z 927.589,A -85,B 0,C 180,E1 18210.717,E2 18210.717} C_VEL
LIN {X 0,Y 452.013,Z 996.513,A -85,B 0,C 180,E1 18214.713,E2 18214.713} C_VEL
LIN {X 0,Y 426.766,Z 1061.584,A -85,B 0,C 180,E1 18220.858,E2 18220.858} C_VEL
LIN {X 0,Y 402.002,Z 1117.953,A -85,B 0,C 180,E1 18229.4,E2 18229.4} C_VEL
LIN {X 0,Y 383.719,Z 1160.762,A -85,B 0,C 180,E1 18239.739,E2 18239.739} C_VEL
LIN {X 0,Y 373.899,Z 1189.47,A -85,B 0,C 180,E1 18251.064,E2 18251.064} C_VEL
LIN {X 0,Y 371.354,Z 1203.89,A -85,B 0,C 180,E1 18261.78,E2 18261.78} C_VEL
LIN {X 0,Y 371.091,Z 1207.191,A -85,B 0,C 180,E1 18271.168,E2 18271.168} C_VEL
LIN {X 0,Y 371.812,Z 1200.296,A -85,B 0,C 180,E1 18281.868,E2 18281.868} C_VEL
LIN {X 0,Y 375.882,Z 1181.949,A -85,B 0,C 180,E1 18292.535,E2 18292.535} C_VEL
LIN {X 0,Y 388.134,Z 1149.246,A -85,B 0,C 180,E1 18303.552,E2 18303.552} C_VEL
LIN {X 0,Y 409.341,Z 1101.319,A -85,B 0,C 180,E1 18313.563,E2 18313.563} C_VEL
LIN {X 0,Y 417.817,Z 1082.444,A -85,B 0,C 180,E1 18316.441,E2 18316.441} C_VEL
LIN {X 0,Y 421.955,Z 1059.979,A -85,B 0,C 180,E1 18320.151,E2 18320.151} C_VEL
LIN {X 0,Y 447.694,Z 994.865,A -85,B 0,C 180,E1 18326.279,E2 18326.279} C_VEL
LIN {X 0,Y 467.693,Z 927.484,A -85,B 0,C 180,E1 18330.289,E2 18330.289} C_VEL
LIN {X 0,Y 453.343,Z 887.247,A -85,B 0,C 180,E1 18337.399,E2 18337.399} C_VEL
LIN {X 0,Y 437.577,Z 856.601,A -85,B 0,C 180,E1 18345.927,E2 18345.927} C_VEL
LIN {X 0,Y 428.03,Z 839.945,A -85,B 0,C 180,E1 18354.128,E2 18354.128} C_VEL
LIN {X 0,Y 425.413,Z 833.757,A -85,B 0,C 180,E1 18363.239,E2 18363.239} C_VEL
LIN {X 0,Y 432.392,Z 846.855,A -85,B 0,C 180,E1 18373.814,E2 18373.814} C_VEL
LIN {X 0,Y 447.969,Z 874.632,A -85,B 0,C 180,E1 18383.306,E2 18383.306} C_VEL
LIN {X 0,Y 463.33,Z 910.129,A -85,B 0,C 180,E1 18390.648,E2 18390.648} C_VEL
LIN {X 0,Y 467.711,Z 927.579,A -85,B 0,C 180,E1 18393.217,E2 18393.217} C_VEL
LIN {X 0,Y 446.142,Z 995.72,A -85,B 0,C 180,E1 18397.216,E2 18397.216} C_VEL
LIN {X 0,Y 419.908,Z 1057.887,A -85,B 0,C 180,E1 18403.351,E2 18403.351} C_VEL
LIN {X 0,Y 395.027,Z 1108.823,A -85,B 0,C 180,E1 18411.646,E2 18411.646} C_VEL
LIN {X 0,Y 376.34,Z 1146.717,A -85,B 0,C 180,E1 18421.742,E2 18421.742} C_VEL
LIN {X 0,Y 366.073,Z 1171.676,A -85,B 0,C 180,E1 18433.145,E2 18433.145} C_VEL
LIN {X 0,Y 363.402,Z 1183.073,A -85,B 0,C 180,E1 18444.014,E2 18444.014} C_VEL
LIN {X 0,Y 363.257,Z 1184.009,A -85,B 0,C 180,E1 18453.593,E2 18453.593} C_VEL
LIN {X 0,Y 365.151,Z 1175.065,A -85,B 0,C 180,E1 18464.432,E2 18464.432} C_VEL
LIN {X 0,Y 373.505,Z 1152.291,A -85,B 0,C 180,E1 18476.186,E2 18476.186} C_VEL
LIN {X 0,Y 391.486,Z 1115.294,A -85,B 0,C 180,E1 18486.903,E2 18486.903} C_VEL
LIN {X 0,Y 416.229,Z 1065.587,A -85,B 0,C 180,E1 18495.53,E2 18495.53} C_VEL
LIN {X 0,Y 441.958,Z 1006.056,A -85,B 0,C 180,E1 18501.868,E2 18501.868} C_VEL
LIN {X 0,Y 464.998,Z 936.8,A -85,B 0,C 180,E1 18506.271,E2 18506.271} C_VEL
LIN {X 0,Y 467.585,Z 923.485,A -85,B 0,C 180,E1 18507.062,E2 18507.062} C_VEL
LIN {X 0,Y 451.258,Z 881.443,A -85,B 0,C 180,E1 18514.882,E2 18514.882} C_VEL
LIN {X 0,Y 435.489,Z 852.3,A -85,B 0,C 180,E1 18523.635,E2 18523.635} C_VEL
LIN {X 0,Y 427.318,Z 839.215,A -85,B 0,C 180,E1 18531.081,E2 18531.081} C_VEL
LIN {X 0,Y 425.112,Z 833.461,A -85,B 0,C 180,E1 18539.382,E2 18539.382} C_VEL
LIN {X 0,Y 432.261,Z 846.859,A -85,B 0,C 180,E1 18550.324,E2 18550.324} C_VEL
LIN {X 0,Y 447.467,Z 875.072,A -85,B 0,C 180,E1 18559.743,E2 18559.743} C_VEL
LIN {X 0,Y 462.944,Z 912.772,A -85,B 0,C 180,E1 18567.344,E2 18567.344} C_VEL
LIN {X 0,Y 467.447,Z 931.409,A -85,B 0,C 180,E1 18570.052,E2 18570.052} C_VEL
LIN {X 0,Y 445.387,Z 1001.572,A -85,B 0,C 180,E1 18574.239,E2 18574.239} C_VEL
LIN {X 0,Y 419.322,Z 1065.811,A -85,B 0,C 180,E1 18580.543,E2 18580.543} C_VEL
LIN {X 0,Y 393.936,Z 1121.188,A -85,B 0,C 180,E1 18589.316,E2 18589.316} C_VEL
LIN {X 0,Y 374.861,Z 1164.133,A -85,B 0,C 180,E1 18600.295,E2 18600.295} C_VEL
LIN {X 0,Y 365.473,Z 1191.369,A -85,B 0,C 180,E1 18611.865,E2 18611.865} C_VEL
LIN {X 0,Y 363.354,Z 1203.637,A -85,B 0,C 180,E1 18621.598,E2 18621.598} C_VEL
LIN {X 0,Y 363.09,Z 1206.944,A -85,B 0,C 180,E1 18631.194,E2 18631.194} C_VEL
LIN {X 0,Y 363.849,Z 1200.231,A -85,B 0,C 180,E1 18641.949,E2 18641.949} C_VEL
LIN {X 0,Y 368.219,Z 1181.675,A -85,B 0,C 180,E1 18653.03,E2 18653.03} C_VEL
LIN {X 0,Y 381.02,Z 1149.141,A -85,B 0,C 180,E1 18664.205,E2 18664.205} C_VEL
LIN {X 0,Y 403.202,Z 1101.156,A -85,B 0,C 180,E1 18674.361,E2 18674.361} C_VEL
LIN {X 0,Y 421.955,Z 1059.979,A -85,B 0,C 180,E1 18680.151,E2 18680.151} C_VEL
LIN {X 0,Y 426.916,Z 1036,A -85,B 0,C 180,E1 18683.621,E2 18683.621} C_VEL
LIN {X 0,Y 452.038,Z 969.299,A -85,B 0,C 180,E1 18688.809,E2 18688.809} C_VEL
LIN {X 0,Y 462.493,Z 930.889,A -85,B 0,C 180,E1 18691.029,E2 18691.029} C_VEL
LIN {X 0,Y 448.952,Z 891.566,A -85,B 0,C 180,E1 18698.262,E2 18698.262} C_VEL
LIN {X 0,Y 433.486,Z 860.355,A -85,B 0,C 180,E1 18707.467,E2 18707.467} C_VEL
LIN {X 0,Y 425.211,Z 846.44,A -85,B 0,C 180,E1 18715.885,E2 18715.885} C_VEL
LIN {X 0,Y 424.01,Z 841.66,A -85,B 0,C 180,E1 18723.157,E2 18723.157} C_VEL
LIN {X 0,Y 430.576,Z 854.519,A -85,B 0,C 180,E1 18733.614,E2 18733.614} C_VEL
LIN {X 0,Y 445.271,Z 882.262,A -85,B 0,C 180,E1 18743.186,E2 18743.186} C_VEL
LIN {X 0,Y 459.969,Z 918.818,A -85,B 0,C 180,E1 18750.739,E2 18750.739} C_VEL
LIN {X 0,Y 462.399,Z 931.855,A -85,B 0,C 180,E1 18752.561,E2 18752.561} C_VEL
LIN {X 0,Y 439.982,Z 999.415,A -85,B 0,C 180,E1 18756.637,E2 18756.637} C_VEL
LIN {X 0,Y 413.547,Z 1059.795,A -85,B 0,C 180,E1 18762.735,E2 18762.735} C_VEL
LIN {X 0,Y 388.061,Z 1110.125,A -85,B 0,C 180,E1 18771.11,E2 18771.11} C_VEL
LIN {X 0,Y 368.259,Z 1148.669,A -85,B 0,C 180,E1 18781.736,E2 18781.736} C_VEL
LIN {X 0,Y 357.558,Z 1173.784,A -85,B 0,C 180,E1 18794,E2 18794} C_VEL
LIN {X 0,Y 355.421,Z 1183.321,A -85,B 0,C 180,E1 18803.879,E2 18803.879} C_VEL
LIN {X 0,Y 355.277,Z 1184.256,A -85,B 0,C 180,E1 18813.673,E2 18813.673} C_VEL
LIN {X 0,Y 357.276,Z 1175.319,A -85,B 0,C 180,E1 18824.757,E2 18824.757} C_VEL
LIN {X 0,Y 365.832,Z 1153.161,A -85,B 0,C 180,E1 18836.508,E2 18836.508} C_VEL
LIN {X 0,Y 384.29,Z 1116.832,A -85,B 0,C 180,E1 18847.357,E2 18847.357} C_VEL
LIN {X 0,Y 409.929,Z 1067.202,A -85,B 0,C 180,E1 18856.173,E2 18856.173} C_VEL
LIN {X 0,Y 436.695,Z 1007.287,A -85,B 0,C 180,E1 18862.634,E2 18862.634} C_VEL
LIN {X 0,Y 460.511,Z 937.755,A -85,B 0,C 180,E1 18867.079,E2 18867.079} C_VEL
LIN {X 0,Y 462.121,Z 926.274,A -85,B 0,C 180,E1 18867.937,E2 18867.937} C_VEL
LIN {X 0,Y 447.069,Z 886.301,A -85,B 0,C 180,E1 18875.691,E2 18875.691} C_VEL
LIN {X 0,Y 432.599,Z 858.629,A -85,B 0,C 180,E1 18884.43,E2 18884.43} C_VEL
LIN {X 0,Y 425.625,Z 846.917,A -85,B 0,C 180,E1 18891.304,E2 18891.304} C_VEL
LIN {X 0,Y 423.71,Z 841.48,A -85,B 0,C 180,E1 18899.38,E2 18899.38} C_VEL
LIN {X 0,Y 430.325,Z 854.413,A -85,B 0,C 180,E1 18910.05,E2 18910.05} C_VEL
LIN {X 0,Y 444.605,Z 882.511,A -85,B 0,C 180,E1 18919.565,E2 18919.565} C_VEL
LIN {X 0,Y 459.142,Z 920.51,A -85,B 0,C 180,E1 18927.268,E2 18927.268} C_VEL
LIN {X 0,Y 461.87,Z 935.936,A -85,B 0,C 180,E1 18929.406,E2 18929.406} C_VEL
LIN {X 0,Y 439.775,Z 1003.644,A -85,B 0,C 180,E1 18933.543,E2 18933.543} C_VEL
LIN {X 0,Y 412.928,Z 1067.536,A -85,B 0,C 180,E1 18939.929,E2 18939.929} C_VEL
LIN {X 0,Y 386.826,Z 1122.374,A -85,B 0,C 180,E1 18948.814,E2 18948.814} C_VEL
LIN {X 0,Y 366.997,Z 1165.197,A -85,B 0,C 180,E1 18960.105,E2 18960.105} C_VEL
LIN {X 0,Y 357.658,Z 1191.104,A -85,B 0,C 180,E1 18971.455,E2 18971.455} C_VEL
LIN {X 0,Y 355.387,Z 1203.386,A -85,B 0,C 180,E1 18981.408,E2 18981.408} C_VEL
LIN {X 0,Y 355.093,Z 1206.697,A -85,B 0,C 180,E1 18991.221,E2 18991.221} C_VEL
LIN {X 0,Y 355.876,Z 1199.895,A -85,B 0,C 180,E1 19002.3,E2 19002.3} C_VEL
LIN {X 0,Y 360.556,Z 1181.401,A -85,B 0,C 180,E1 19013.549,E2 19013.549} C_VEL
LIN {X 0,Y 374.102,Z 1148.847,A -85,B 0,C 180,E1 19024.928,E2 19024.928} C_VEL
LIN {X 0,Y 396.644,Z 1102.018,A -85,B 0,C 180,E1 19035.014,E2 19035.014} C_VEL
LIN {X 0,Y 424.126,Z 1042.348,A -85,B 0,C 180,E1 19042.972,E2 19042.972} C_VEL
LIN {X 0,Y 426.916,Z 1036,A -85,B 0,C 180,E1 19043.621,E2 19043.621} C_VEL
LIN {X 0,Y 432.371,Z 1010.358,A -85,B 0,C 180,E1 19046.819,E2 19046.819} C_VEL
LIN {X 0,Y 457.033,Z 938.795,A -85,B 0,C 180,E1 19051.323,E2 19051.323} C_VEL
LIN {X 0,Y 449.522,Z 908.705,A -85,B 0,C 180,E1 19056.34,E2 19056.34} C_VEL
LIN {X 0,Y 435.165,Z 875.827,A -85,B 0,C 180,E1 19064.814,E2 19064.814} C_VEL
LIN {X 0,Y 424.999,Z 855.644,A -85,B 0,C 180,E1 19074.086,E2 19074.086} C_VEL
LIN {X 0,Y 422.476,Z 849.549,A -85,B 0,C 180,E1 19083.068,E2 19083.068} C_VEL
LIN {X 0,Y 428.477,Z 862.19,A -85,B 0,C 180,E1 19093.421,E2 19093.421} C_VEL
LIN {X 0,Y 442.286,Z 889.415,A -85,B 0,C 180,E1 19102.926,E2 19102.926} C_VEL
LIN {X 0,Y 455.889,Z 925.552,A -85,B 0,C 180,E1 19110.49,E2 19110.49} C_VEL
LIN {X 0,Y 457.296,Z 935.328,A -85,B 0,C 180,E1 19111.855,E2 19111.855} C_VEL
LIN {X 0,Y 434.252,Z 1002.17,A -85,B 0,C 180,E1 19115.975,E2 19115.975} C_VEL
LIN {X 0,Y 406.454,Z 1063.325,A -85,B 0,C 180,E1 19122.322,E2 19122.322} C_VEL
LIN {X 0,Y 380.171,Z 1113.146,A -85,B 0,C 180,E1 19130.926,E2 19130.926} C_VEL
LIN {X 0,Y 360.312,Z 1150.346,A -85,B 0,C 180,E1 19141.63,E2 19141.63} C_VEL
LIN {X 0,Y 349.772,Z 1174.038,A -85,B 0,C 180,E1 19153.634,E2 19153.634} C_VEL
LIN {X 0,Y 347.427,Z 1183.569,A -85,B 0,C 180,E1 19163.738,E2 19163.738} C_VEL
LIN {X 0,Y 347.274,Z 1184.505,A -85,B 0,C 180,E1 19173.758,E2 19173.758} C_VEL
LIN {X 0,Y 349.403,Z 1175.574,A -85,B 0,C 180,E1 19185.097,E2 19185.097} C_VEL
LIN {X 0,Y 358.465,Z 1153.427,A -85,B 0,C 180,E1 19197.097,E2 19197.097} C_VEL
LIN {X 0,Y 377.731,Z 1117.117,A -85,B 0,C 180,E1 19208.12,E2 19208.12} C_VEL
LIN {X 0,Y 404.316,Z 1067.534,A -85,B 0,C 180,E1 19217.008,E2 19217.008} C_VEL
LIN {X 0,Y 431.902,Z 1007.53,A -85,B 0,C 180,E1 19223.5,E2 19223.5} C_VEL
LIN {X 0,Y 456.321,Z 937.971,A -85,B 0,C 180,E1 19227.939,E2 19227.939} C_VEL
LIN {X 0,Y 456.896,Z 929.506,A -85,B 0,C 180,E1 19228.755,E2 19228.755} C_VEL
LIN {X 0,Y 442.713,Z 890.51,A -85,B 0,C 180,E1 19236.664,E2 19236.664} C_VEL
LIN {X 0,Y 429.398,Z 864.352,A -85,B 0,C 180,E1 19245.446,E2 19245.446} C_VEL
LIN {X 0,Y 423.77,Z 854.386,A -85,B 0,C 180,E1 19251.784,E2 19251.784} C_VEL
LIN {X 0,Y 422.179,Z 849.422,A -85,B 0,C 180,E1 19259.377,E2 19259.377} C_VEL
LIN {X 0,Y 428.26,Z 862.18,A -85,B 0,C 180,E1 19269.922,E2 19269.922} C_VEL
LIN {X 0,Y 441.607,Z 889.715,A -85,B 0,C 180,E1 19279.312,E2 19279.312} C_VEL
LIN {X 0,Y 455.059,Z 927.513,A -85,B 0,C 180,E1 19287.052,E2 19287.052} C_VEL
LIN {X 0,Y 456.379,Z 940.524,A -85,B 0,C 180,E1 19288.757,E2 19288.757} C_VEL
LIN {X 0,Y 432.529,Z 1010.048,A -85,B 0,C 180,E1 19293.189,E2 19293.189} C_VEL
LIN {X 0,Y 404.67,Z 1073.147,A -85,B 0,C 180,E1 19299.8,E2 19299.8} C_VEL
LIN {X 0,Y 378.068,Z 1126.821,A -85,B 0,C 180,E1 19308.981,E2 19308.981} C_VEL
LIN {X 0,Y 358.687,Z 1167.166,A -85,B 0,C 180,E1 19320.216,E2 19320.216} C_VEL
LIN {X 0,Y 349.473,Z 1192.167,A -85,B 0,C 180,E1 19331.866,E2 19331.866} C_VEL
LIN {X 0,Y 347.393,Z 1203.134,A -85,B 0,C 180,E1 19341.209,E2 19341.209} C_VEL
LIN {X 0,Y 347.092,Z 1206.449,A -85,B 0,C 180,E1 19351.249,E2 19351.249} C_VEL
LIN {X 0,Y 347.904,Z 1199.639,A -85,B 0,C 180,E1 19362.586,E2 19362.586} C_VEL
LIN {X 0,Y 352.933,Z 1181.129,A -85,B 0,C 180,E1 19374.089,E2 19374.089} C_VEL
LIN {X 0,Y 367.259,Z 1148.556,A -85,B 0,C 180,E1 19385.677,E2 19385.677} C_VEL
LIN {X 0,Y 390.74,Z 1101.696,A -85,B 0,C 180,E1 19395.887,E2 19395.887} C_VEL
LIN {X 0,Y 418.943,Z 1042.452,A -85,B 0,C 180,E1 19403.833,E2 19403.833} C_VEL
LIN {X 0,Y 432.371,Z 1010.358,A -85,B 0,C 180,E1 19406.819,E2 19406.819} C_VEL
LIN {X 0,Y 438.425,Z 983.172,A -85,B 0,C 180,E1 19409.709,E2 19409.709} C_VEL
LIN {X 0,Y 452.271,Z 938.727,A -85,B 0,C 180,E1 19412.37,E2 19412.37} C_VEL
LIN {X 0,Y 440.806,Z 902.284,A -85,B 0,C 180,E1 19419.575,E2 19419.575} C_VEL
LIN {X 0,Y 428.323,Z 874.474,A -85,B 0,C 180,E1 19428.356,E2 19428.356} C_VEL
LIN {X 0,Y 421.604,Z 861.706,A -85,B 0,C 180,E1 19436.367,E2 19436.367} C_VEL
LIN {X 0,Y 420.847,Z 857.572,A -85,B 0,C 180,E1 19443.08,E2 19443.08} C_VEL
LIN {X 0,Y 426.376,Z 869.932,A -85,B 0,C 180,E1 19453.282,E2 19453.282} C_VEL
LIN {X 0,Y 439.255,Z 896.648,A -85,B 0,C 180,E1 19462.711,E2 19462.711} C_VEL
LIN {X 0,Y 452.049,Z 933.463,A -85,B 0,C 180,E1 19470.469,E2 19470.469} C_VEL
LIN {X 0,Y 451.145,Z 942.617,A -85,B 0,C 180,E1 19471.317,E2 19471.317} C_VEL
LIN {X 0,Y 426.893,Z 1008.86,A -85,B 0,C 180,E1 19475.605,E2 19475.605} C_VEL
LIN {X 0,Y 398.543,Z 1068.436,A -85,B 0,C 180,E1 19482.101,E2 19482.101} C_VEL
LIN {X 0,Y 371.341,Z 1117.756,A -85,B 0,C 180,E1 19491.108,E2 19491.108} C_VEL
LIN {X 0,Y 351.35,Z 1153.83,A -85,B 0,C 180,E1 19502.269,E2 19502.269} C_VEL
LIN {X 0,Y 341.333,Z 1175.959,A -85,B 0,C 180,E1 19514.542,E2 19514.542} C_VEL
LIN {X 0,Y 339.229,Z 1184.796,A -85,B 0,C 180,E1 19526.158,E2 19526.158} C_VEL
LIN {X 0,Y 339.383,Z 1183.768,A -85,B 0,C 180,E1 19536.417,E2 19536.417} C_VEL
LIN {X 0,Y 342.873,Z 1171.729,A -85,B 0,C 180,E1 19548.445,E2 19548.445} C_VEL
LIN {X 0,Y 355.463,Z 1145.597,A -85,B 0,C 180,E1 19560.79,E2 19560.79} C_VEL
LIN {X 0,Y 377.973,Z 1105.789,A -85,B 0,C 180,E1 19571.457,E2 19571.457} C_VEL
LIN {X 0,Y 406.564,Z 1052.467,A -85,B 0,C 180,E1 19579.88,E2 19579.88} C_VEL
LIN {X 0,Y 434.491,Z 990.094,A -85,B 0,C 180,E1 19585.734,E2 19585.734} C_VEL
LIN {X 0,Y 452.247,Z 935.178,A -85,B 0,C 180,E1 19589.158,E2 19589.158} C_VEL
LIN {X 0,Y 439.945,Z 898.738,A -85,B 0,C 180,E1 19596.647,E2 19596.647} C_VEL
LIN {X 0,Y 427.305,Z 872.122,A -85,B 0,C 180,E1 19605.559,E2 19605.559} C_VEL
LIN {X 0,Y 421.819,Z 862.027,A -85,B 0,C 180,E1 19612.006,E2 19612.006} C_VEL
LIN {X 0,Y 420.568,Z 857.362,A -85,B 0,C 180,E1 19619.375,E2 19619.375} C_VEL
LIN {X 0,Y 426.073,Z 869.726,A -85,B 0,C 180,E1 19629.706,E2 19629.706} C_VEL
LIN {X 0,Y 438.121,Z 896.001,A -85,B 0,C 180,E1 19638.835,E2 19638.835} C_VEL
LIN {X 0,Y 450.443,Z 932.675,A -85,B 0,C 180,E1 19646.541,E2 19646.541} C_VEL
LIN {X 0,Y 451.198,Z 944.234,A -85,B 0,C 180,E1 19648.048,E2 19648.048} C_VEL
LIN {X 0,Y 426.234,Z 1014.087,A -85,B 0,C 180,E1 19652.625,E2 19652.625} C_VEL
LIN {X 0,Y 397.434,Z 1076.729,A -85,B 0,C 180,E1 19659.4,E2 19659.4} C_VEL
LIN {X 0,Y 369.948,Z 1129.969,A -85,B 0,C 180,E1 19668.879,E2 19668.879} C_VEL
LIN {X 0,Y 349.843,Z 1170.277,A -85,B 0,C 180,E1 19680.81,E2 19680.81} C_VEL
LIN {X 0,Y 341.044,Z 1194.602,A -85,B 0,C 180,E1 19693.197,E2 19693.197} C_VEL
LIN {X 0,Y 339.163,Z 1204.606,A -85,B 0,C 180,E1 19703.579,E2 19703.579} C_VEL
LIN {X 0,Y 339.107,Z 1205.703,A -85,B 0,C 180,E1 19713.844,E2 19713.844} C_VEL
LIN {X 0,Y 340.527,Z 1196.266,A -85,B 0,C 180,E1 19725.495,E2 19725.495} C_VEL
LIN {X 0,Y 349.439,Z 1171.922,A -85,B 0,C 180,E1 19738.512,E2 19738.512} C_VEL
LIN {X 0,Y 368.97,Z 1132.198,A -85,B 0,C 180,E1 19750.572,E2 19750.572} C_VEL
LIN {X 0,Y 395.646,Z 1080.63,A -85,B 0,C 180,E1 19760.046,E2 19760.046} C_VEL
LIN {X 0,Y 424.61,Z 1018.151,A -85,B 0,C 180,E1 19767.064,E2 19767.064} C_VEL
LIN {X 0,Y 438.425,Z 983.172,A -85,B 0,C 180,E1 19769.709,E2 19769.709} C_VEL
LIN {X 0,Y 444.197,Z 954.443,A -85,B 0,C 180,E1 19772.31,E2 19772.31} C_VEL
LIN {X 0,Y 447.025,Z 941.595,A -85,B 0,C 180,E1 19773.242,E2 19773.242} C_VEL
LIN {X 0,Y 436.115,Z 906.013,A -85,B 0,C 180,E1 19780.672,E2 19780.672} C_VEL
LIN {X 0,Y 424.803,Z 880.043,A -85,B 0,C 180,E1 19789.461,E2 19789.461} C_VEL
LIN {X 0,Y 419.409,Z 868.784,A -85,B 0,C 180,E1 19797.127,E2 19797.127} C_VEL
LIN {X 0,Y 418.955,Z 865.474,A -85,B 0,C 180,E1 19803.094,E2 19803.094} C_VEL
LIN {X 0,Y 424.155,Z 877.741,A -85,B 0,C 180,E1 19813.165,E2 19813.165} C_VEL
LIN {X 0,Y 435.299,Z 902.331,A -85,B 0,C 180,E1 19822.046,E2 19822.046} C_VEL
LIN {X 0,Y 446.968,Z 937.399,A -85,B 0,C 180,E1 19829.734,E2 19829.734} C_VEL
LIN {X 0,Y 446.477,Z 945.045,A -85,B 0,C 180,E1 19830.529,E2 19830.529} C_VEL
LIN {X 0,Y 420.933,Z 1012.283,A -85,B 0,C 180,E1 19834.957,E2 19834.957} C_VEL
LIN {X 0,Y 391.111,Z 1072.288,A -85,B 0,C 180,E1 19841.723,E2 19841.723} C_VEL
LIN {X 0,Y 363.128,Z 1120.941,A -85,B 0,C 180,E1 19851.015,E2 19851.015} C_VEL
LIN {X 0,Y 342.292,Z 1157.252,A -85,B 0,C 180,E1 19862.994,E2 19862.994} C_VEL
LIN {X 0,Y 332.956,Z 1177.709,A -85,B 0,C 180,E1 19875.495,E2 19875.495} C_VEL
LIN {X 0,Y 331.23,Z 1185.044,A -85,B 0,C 180,E1 19886.065,E2 19886.065} C_VEL
LIN {X 0,Y 331.393,Z 1184.017,A -85,B 0,C 180,E1 19896.572,E2 19896.572} C_VEL
LIN {X 0,Y 335.173,Z 1171.83,A -85,B 0,C 180,E1 19909.001,E2 19909.001} C_VEL
LIN {X 0,Y 348.859,Z 1145.167,A -85,B 0,C 180,E1 19921.742,E2 19921.742} C_VEL
LIN {X 0,Y 372.663,Z 1104.645,A -85,B 0,C 180,E1 19932.582,E2 19932.582} C_VEL
LIN {X 0,Y 402.073,Z 1051.431,A -85,B 0,C 180,E1 19940.931,E2 19940.931} C_VEL
LIN {X 0,Y 430.584,Z 989.117,A -85,B 0,C 180,E1 19946.718,E2 19946.718} C_VEL
LIN {X 0,Y 447.263,Z 939.245,A -85,B 0,C 180,E1 19949.843,E2 19949.843} C_VEL
LIN {X 0,Y 435.739,Z 903.481,A -85,B 0,C 180,E1 19957.491,E2 19957.491} C_VEL
LIN {X 0,Y 423.909,Z 876.651,A -85,B 0,C 180,E1 19966.959,E2 19966.959} C_VEL
LIN {X 0,Y 418.757,Z 864.931,A -85,B 0,C 180,E1 19976.994,E2 19976.994} C_VEL
LIN {X 0,Y 422.123,Z 874.614,A -85,B 0,C 180,E1 19987.708,E2 19987.708} C_VEL
LIN {X 0,Y 431.138,Z 894.099,A -85,B 0,C 180,E1 19995.932,E2 19995.932} C_VEL
LIN {X 0,Y 442.366,Z 925.333,A -85,B 0,C 180,E1 20003.661,E2 20003.661} C_VEL
LIN {X 0,Y 446.378,Z 947.022,A -85,B 0,C 180,E1 20007.281,E2 20007.281} C_VEL
LIN {X 0,Y 420.784,Z 1016.163,A -85,B 0,C 180,E1 20011.881,E2 20011.881} C_VEL
LIN {X 0,Y 390.803,Z 1079.069,A -85,B 0,C 180,E1 20018.82,E2 20018.82} C_VEL
LIN {X 0,Y 362.407,Z 1131.81,A -85,B 0,C 180,E1 20028.522,E2 20028.522} C_VEL
LIN {X 0,Y 342.388,Z 1170.311,A -85,B 0,C 180,E1 20040.252,E2 20040.252} C_VEL
LIN {X 0,Y 333.148,Z 1194.341,A -85,B 0,C 180,E1 20052.787,E2 20052.787} C_VEL
LIN {X 0,Y 331.16,Z 1204.356,A -85,B 0,C 180,E1 20063.423,E2 20063.423} C_VEL
LIN {X 0,Y 331.113,Z 1205.956,A -85,B 0,C 180,E1 20071.31,E2 20071.31} C_VEL
LIN {X 0,Y 331.797,Z 1200.407,A -85,B 0,C 180,E1 20081.866,E2 20081.866} C_VEL
LIN {X 0,Y 337.246,Z 1181.983,A -85,B 0,C 180,E1 20094.576,E2 20094.576} C_VEL
LIN {X 0,Y 352.516,Z 1150.315,A -85,B 0,C 180,E1 20106.612,E2 20106.612} C_VEL
LIN {X 0,Y 378.446,Z 1102.495,A -85,B 0,C 180,E1 20117.469,E2 20117.469} C_VEL
LIN {X 0,Y 408.289,Z 1043.884,A -85,B 0,C 180,E1 20125.494,E2 20125.494} C_VEL
LIN {X 0,Y 436.315,Z 977.15,A -85,B 0,C 180,E1 20130.997,E2 20130.997} C_VEL
LIN {X 0,Y 444.197,Z 954.443,A -85,B 0,C 180,E1 20132.31,E2 20132.31} C_VEL
LIN {X 0,Y 443.612,Z 942.785,A -85,B 0,C 180,E1 20133.935,E2 20133.935} C_VEL
LIN {X 0,Y 439.389,Z 934.092,A -85,B 0,C 180,E1 20136.111,E2 20136.111} C_VEL
LIN {X 0,Y 428.507,Z 902.235,A -85,B 0,C 180,E1 20144.046,E2 20144.046} C_VEL
LIN {X 0,Y 419.724,Z 881.734,A -85,B 0,C 180,E1 20152.773,E2 20152.773} C_VEL
LIN {X 0,Y 417.125,Z 872.872,A -85,B 0,C 180,E1 20162.716,E2 20162.716} C_VEL
LIN {X 0,Y 421.722,Z 885.425,A -85,B 0,C 180,E1 20173.044,E2 20173.044} C_VEL
LIN {X 0,Y 432.658,Z 910.798,A -85,B 0,C 180,E1 20182.187,E2 20182.187} C_VEL
LIN {X 0,Y 442.679,Z 944.122,A -85,B 0,C 180,E1 20189.507,E2 20189.507} C_VEL
LIN {X 0,Y 416.36,Z 1012.663,A -85,B 0,C 180,E1 20194.046,E2 20194.046} C_VEL
LIN {X 0,Y 386.736,Z 1070.873,A -85,B 0,C 180,E1 20200.561,E2 20200.561} C_VEL
LIN {X 0,Y 358.299,Z 1118.889,A -85,B 0,C 180,E1 20209.602,E2 20209.602} C_VEL
LIN {X 0,Y 336.766,Z 1154.542,A -85,B 0,C 180,E1 20221.05,E2 20221.05} C_VEL
LIN {X 0,Y 325.7,Z 1176.464,A -85,B 0,C 180,E1 20233.78,E2 20233.78} C_VEL
LIN {X 0,Y 323.231,Z 1185.292,A -85,B 0,C 180,E1 20245.967,E2 20245.967} C_VEL
LIN {X 0,Y 323.418,Z 1184.266,A -85,B 0,C 180,E1 20256.735,E2 20256.735} C_VEL
LIN {X 0,Y 327.125,Z 1172.808,A -85,B 0,C 180,E1 20268.937,E2 20268.937} C_VEL
LIN {X 0,Y 340.824,Z 1147.08,A -85,B 0,C 180,E1 20281.845,E2 20281.845} C_VEL
LIN {X 0,Y 365.816,Z 1106.375,A -85,B 0,C 180,E1 20293.162,E2 20293.162} C_VEL
LIN {X 0,Y 396.275,Z 1053.151,A -85,B 0,C 180,E1 20301.68,E2 20301.68} C_VEL
LIN {X 0,Y 425.432,Z 991.457,A -85,B 0,C 180,E1 20307.492,E2 20307.492} C_VEL
LIN {X 0,Y 442.383,Z 943.807,A -85,B 0,C 180,E1 20310.472,E2 20310.472} C_VEL
LIN {X 0,Y 431.567,Z 908.401,A -85,B 0,C 180,E1 20318.351,E2 20318.351} C_VEL
LIN {X 0,Y 420.917,Z 883.478,A -85,B 0,C 180,E1 20327.659,E2 20327.659} C_VEL
LIN {X 0,Y 416.85,Z 872.66,A -85,B 0,C 180,E1 20337.413,E2 20337.413} C_VEL
LIN {X 0,Y 419.992,Z 882.727,A -85,B 0,C 180,E1 20347.901,E2 20347.901} C_VEL
LIN {X 0,Y 428.993,Z 903.751,A -85,B 0,C 180,E1 20356.464,E2 20356.464} C_VEL
LIN {X 0,Y 439.42,Z 936.109,A -85,B 0,C 180,E1 20364.21,E2 20364.21} C_VEL
LIN {X 0,Y 441.247,Z 950.865,A -85,B 0,C 180,E1 20366.56,E2 20366.56} C_VEL
LIN {X 0,Y 414.698,Z 1019.715,A -85,B 0,C 180,E1 20371.253,E2 20371.253} C_VEL
LIN {X 0,Y 384.024,Z 1081.539,A -85,B 0,C 180,E1 20378.263,E2 20378.263} C_VEL
LIN {X 0,Y 354.954,Z 1133.518,A -85,B 0,C 180,E1 20388.117,E2 20388.117} C_VEL
LIN {X 0,Y 334.282,Z 1171.734,A -85,B 0,C 180,E1 20400.255,E2 20400.255} C_VEL
LIN {X 0,Y 324.951,Z 1195.263,A -85,B 0,C 180,E1 20413.337,E2 20413.337} C_VEL
LIN {X 0,Y 323.17,Z 1204.107,A -85,B 0,C 180,E1 20423.26,E2 20423.26} C_VEL
LIN {X 0,Y 323.131,Z 1205.709,A -85,B 0,C 180,E1 20431.342,E2 20431.342} C_VEL
LIN {X 0,Y 323.823,Z 1200.153,A -85,B 0,C 180,E1 20442.163,E2 20442.163} C_VEL
LIN {X 0,Y 329.142,Z 1183.083,A -85,B 0,C 180,E1 20454.496,E2 20454.496} C_VEL
LIN {X 0,Y 345.643,Z 1150.32,A -85,B 0,C 180,E1 20467.358,E2 20467.358} C_VEL
LIN {X 0,Y 372.297,Z 1103.081,A -85,B 0,C 180,E1 20478.27,E2 20478.27} C_VEL
LIN {X 0,Y 403.073,Z 1044.686,A -85,B 0,C 180,E1 20486.345,E2 20486.345} C_VEL
LIN {X 0,Y 431.756,Z 978.35,A -85,B 0,C 180,E1 20491.848,E2 20491.848} C_VEL
LIN {X 0,Y 442.139,Z 945.933,A -85,B 0,C 180,E1 20493.891,E2 20493.891} C_VEL
LIN {X 0,Y 439.389,Z 934.092,A -85,B 0,C 180,E1 20496.111,E2 20496.111} C_VEL
LIN {X 0,Y 430.15,Z 922.918,A -85,B 0,C 180,E1 20500.408,E2 20500.408} C_VEL
LIN {X 0,Y 420.427,Z 896.535,A -85,B 0,C 180,E1 20509.053,E2 20509.053} C_VEL
LIN {X 0,Y 415.131,Z 884.081,A -85,B 0,C 180,E1 20517.359,E2 20517.359} C_VEL
LIN {X 0,Y 414.87,Z 881.212,A -85,B 0,C 180,E1 20523.124,E2 20523.124} C_VEL
LIN {X 0,Y 419.204,Z 892.776,A -85,B 0,C 180,E1 20532.791,E2 20532.791} C_VEL
LIN {X 0,Y 429.588,Z 919.08,A -85,B 0,C 180,E1 20542.3,E2 20542.3} C_VEL
LIN {X 0,Y 437.415,Z 949.488,A -85,B 0,C 180,E1 20548.897,E2 20548.897} C_VEL
LIN {X 0,Y 410.658,Z 1015.533,A -85,B 0,C 180,E1 20553.334,E2 20553.334} C_VEL
LIN {X 0,Y 379.347,Z 1074.694,A -85,B 0,C 180,E1 20560.154,E2 20560.154} C_VEL
LIN {X 0,Y 349.669,Z 1122.718,A -85,B 0,C 180,E1 20569.633,E2 20569.633} C_VEL
LIN {X 0,Y 327.678,Z 1157.927,A -85,B 0,C 180,E1 20581.761,E2 20581.761} C_VEL
LIN {X 0,Y 317.254,Z 1178.214,A -85,B 0,C 180,E1 20594.76,E2 20594.76} C_VEL
LIN {X 0,Y 315.234,Z 1185.539,A -85,B 0,C 180,E1 20605.865,E2 20605.865} C_VEL
LIN {X 0,Y 315.431,Z 1184.515,A -85,B 0,C 180,E1 20616.906,E2 20616.906} C_VEL
LIN {X 0,Y 319.396,Z 1173.063,A -85,B 0,C 180,E1 20629.415,E2 20629.415} C_VEL
LIN {X 0,Y 333.413,Z 1148.026,A -85,B 0,C 180,E1 20642.329,E2 20642.329} C_VEL
LIN {X 0,Y 358.981,Z 1107.966,A -85,B 0,C 180,E1 20653.773,E2 20653.773} C_VEL
LIN {X 0,Y 390.181,Z 1055.559,A -85,B 0,C 180,E1 20662.368,E2 20662.368} C_VEL
LIN {X 0,Y 420.281,Z 993.981,A -85,B 0,C 180,E1 20668.271,E2 20668.271} C_VEL
LIN {X 0,Y 437.166,Z 946.85,A -85,B 0,C 180,E1 20671.408,E2 20671.408} C_VEL
LIN {X 0,Y 427.44,Z 913.329,A -85,B 0,C 180,E1 20679.212,E2 20679.212} C_VEL
LIN {X 0,Y 417.854,Z 889.642,A -85,B 0,C 180,E1 20688.63,E2 20688.63} C_VEL
LIN {X 0,Y 414.688,Z 880.535,A -85,B 0,C 180,E1 20699.104,E2 20699.104} C_VEL
LIN {X 0,Y 418.903,Z 892.691,A -85,B 0,C 180,E1 20709.274,E2 20709.274} C_VEL
LIN {X 0,Y 428.336,Z 918.115,A -85,B 0,C 180,E1 20718.316,E2 20718.316} C_VEL
LIN {X 0,Y 436.996,Z 951.596,A -85,B 0,C 180,E1 20725.616,E2 20725.616} C_VEL
LIN {X 0,Y 409.816,Z 1020.633,A -85,B 0,C 180,E1 20730.378,E2 20730.378} C_VEL
LIN {X 0,Y 378.499,Z 1081.853,A -85,B 0,C 180,E1 20737.359,E2 20737.359} C_VEL
LIN {X 0,Y 348.719,Z 1133.223,A -85,B 0,C 180,E1 20747.192,E2 20747.192} C_VEL
LIN {X 0,Y 326.611,Z 1172.252,A -85,B 0,C 180,E1 20759.866,E2 20759.866} C_VEL
LIN {X 0,Y 317.076,Z 1195.005,A -85,B 0,C 180,E1 20772.91,E2 20772.91} C_VEL
LIN {X 0,Y 315.168,Z 1203.858,A -85,B 0,C 180,E1 20783.088,E2 20783.088} C_VEL
LIN {X 0,Y 315.128,Z 1205.462,A -85,B 0,C 180,E1 20791.376,E2 20791.376} C_VEL
LIN {X 0,Y 315.86,Z 1199.899,A -85,B 0,C 180,E1 20802.475,E2 20802.475} C_VEL
LIN {X 0,Y 321.565,Z 1182.818,A -85,B 0,C 180,E1 20815.112,E2 20815.112} C_VEL
LIN {X 0,Y 338.415,Z 1150.978,A -85,B 0,C 180,E1 20827.924,E2 20827.924} C_VEL
LIN {X 0,Y 365.723,Z 1104.602,A -85,B 0,C 180,E1 20838.93,E2 20838.93} C_VEL
LIN {X 0,Y 397.359,Z 1046.668,A -85,B 0,C 180,E1 20847.096,E2 20847.096} C_VEL
LIN {X 0,Y 426.536,Z 981.538,A -85,B 0,C 180,E1 20852.595,E2 20852.595} C_VEL
LIN {X 0,Y 437.256,Z 950.334,A -85,B 0,C 180,E1 20854.538,E2 20854.538} C_VEL
LIN {X 0,Y 430.15,Z 922.918,A -85,B 0,C 180,E1 20860.408,E2 20860.408} C_VEL
LIN {X 0,Y 421.667,Z 915.173,A -85,B 0,C 180,E1 20864.95,E2 20864.95} C_VEL
LIN {X 0,Y 414.489,Z 895.881,A -85,B 0,C 180,E1 20873.671,E2 20873.671} C_VEL
LIN {X 0,Y 412.702,Z 888.539,A -85,B 0,C 180,E1 20882.745,E2 20882.745} C_VEL
LIN {X 0,Y 416.774,Z 901.384,A -85,B 0,C 180,E1 20893.135,E2 20893.135} C_VEL
LIN {X 0,Y 426.544,Z 927.554,A -85,B 0,C 180,E1 20902.468,E2 20902.468} C_VEL
LIN {X 0,Y 432.264,Z 953.635,A -85,B 0,C 180,E1 20908.153,E2 20908.153} C_VEL
LIN {X 0,Y 403.975,Z 1020.521,A -85,B 0,C 180,E1 20912.796,E2 20912.796} C_VEL
LIN {X 0,Y 371.707,Z 1078.971,A -85,B 0,C 180,E1 20919.803,E2 20919.803} C_VEL
LIN {X 0,Y 341.573,Z 1125.787,A -85,B 0,C 180,E1 20929.471,E2 20929.471} C_VEL
LIN {X 0,Y 319.077,Z 1160.428,A -85,B 0,C 180,E1 20942.12,E2 20942.12} C_VEL
LIN {X 0,Y 308.919,Z 1179.937,A -85,B 0,C 180,E1 20955.794,E2 20955.794} C_VEL
LIN {X 0,Y 307.178,Z 1186.252,A -85,B 0,C 180,E1 20968.588,E2 20968.588} C_VEL
LIN {X 0,Y 307.917,Z 1183.13,A -85,B 0,C 180,E1 20979.929,E2 20979.929} C_VEL
LIN {X 0,Y 314.519,Z 1168.196,A -85,B 0,C 180,E1 20993.393,E2 20993.393} C_VEL
LIN {X 0,Y 332.627,Z 1139.221,A -85,B 0,C 180,E1 21006.352,E2 21006.352} C_VEL
LIN {X 0,Y 360.482,Z 1096.979,A -85,B 0,C 180,E1 21016.969,E2 21016.969} C_VEL
LIN {X 0,Y 392.429,Z 1042.94,A -85,B 0,C 180,E1 21024.852,E2 21024.852} C_VEL
LIN {X 0,Y 422.431,Z 979.448,A -85,B 0,C 180,E1 21030.245,E2 21030.245} C_VEL
LIN {X 0,Y 432.275,Z 951.506,A -85,B 0,C 180,E1 21032.021,E2 21032.021} C_VEL
LIN {X 0,Y 423.811,Z 919.871,A -85,B 0,C 180,E1 21039.585,E2 21039.585} C_VEL
LIN {X 0,Y 415.525,Z 897.726,A -85,B 0,C 180,E1 21048.432,E2 21048.432} C_VEL
LIN {X 0,Y 412.472,Z 888.17,A -85,B 0,C 180,E1 21058.967,E2 21058.967} C_VEL
LIN {X 0,Y 416.041,Z 899.746,A -85,B 0,C 180,E1 21068.941,E2 21068.941} C_VEL
LIN {X 0,Y 424.965,Z 925.693,A -85,B 0,C 180,E1 21078.233,E2 21078.233} C_VEL
LIN {X 0,Y 431.999,Z 955.715,A -85,B 0,C 180,E1 21084.923,E2 21084.923} C_VEL
LIN {X 0,Y 403.797,Z 1024.105,A -85,B 0,C 180,E1 21089.712,E2 21089.712} C_VEL
LIN {X 0,Y 371.699,Z 1084.535,A -85,B 0,C 180,E1 21096.789,E2 21096.789} C_VEL
LIN {X 0,Y 341.034,Z 1135.401,A -85,B 0,C 180,E1 21106.861,E2 21106.861} C_VEL
LIN {X 0,Y 319.397,Z 1171.978,A -85,B 0,C 180,E1 21119.112,E2 21119.112} C_VEL
LIN {X 0,Y 309.191,Z 1194.843,A -85,B 0,C 180,E1 21132.547,E2 21132.547} C_VEL
LIN {X 0,Y 307.187,Z 1203.609,A -85,B 0,C 180,E1 21142.908,E2 21142.908} C_VEL
LIN {X 0,Y 307.125,Z 1205.215,A -85,B 0,C 180,E1 21151.412,E2 21151.412} C_VEL
LIN {X 0,Y 307.907,Z 1199.645,A -85,B 0,C 180,E1 21162.802,E2 21162.802} C_VEL
LIN {X 0,Y 314.544,Z 1181.514,A -85,B 0,C 180,E1 21176.297,E2 21176.297} C_VEL
LIN {X 0,Y 333.745,Z 1147.571,A -85,B 0,C 180,E1 21189.754,E2 21189.754} C_VEL
LIN {X 0,Y 362.658,Z 1100.112,A -85,B 0,C 180,E1 21200.675,E2 21200.675} C_VEL
LIN {X 0,Y 395.529,Z 1041.056,A -85,B 0,C 180,E1 21208.668,E2 21208.668} C_VEL
LIN {X 0,Y 425.081,Z 975.162,A -85,B 0,C 180,E1 21213.95,E2 21213.95} C_VEL
LIN {X 0,Y 432.089,Z 953.474,A -85,B 0,C 180,E1 21215.428,E2 21215.428} C_VEL
LIN {X 0,Y 423.966,Z 922.051,A -85,B 0,C 180,E1 21222.799,E2 21222.799} C_VEL
LIN {X 0,Y 421.667,Z 915.173,A -85,B 0,C 180,E1 21224.95,E2 21224.95} C_VEL
LIN {X 0,Y 414.491,Z 910.688,A -85,B 0,C 180,E1 21229.698,E2 21229.698} C_VEL
LIN {X 0,Y 410.283,Z 898.985,A -85,B 0,C 180,E1 21237.858,E2 21237.858} C_VEL
LIN {X 0,Y 410.239,Z 896.73,A -85,B 0,C 180,E1 21243.16,E2 21243.16} C_VEL
LIN {X 0,Y 414.168,Z 909.319,A -85,B 0,C 180,E1 21253.219,E2 21253.219} C_VEL
LIN {X 0,Y 422.656,Z 934.045,A -85,B 0,C 180,E1 21262.129,E2 21262.129} C_VEL
LIN {X 0,Y 426.983,Z 958.423,A -85,B 0,C 180,E1 21267.434,E2 21267.434} C_VEL
LIN {X 0,Y 398.426,Z 1023.313,A -85,B 0,C 180,E1 21272.039,E2 21272.039} C_VEL
LIN {X 0,Y 365.346,Z 1081.171,A -85,B 0,C 180,E1 21279.111,E2 21279.111} C_VEL
LIN {X 0,Y 333.71,Z 1128.452,A -85,B 0,C 180,E1 21289.216,E2 21289.216} C_VEL
LIN {X 0,Y 310.613,Z 1162.443,A -85,B 0,C 180,E1 21302.369,E2 21302.369} C_VEL
LIN {X 0,Y 301.056,Z 1180.188,A -85,B 0,C 180,E1 21315.415,E2 21315.415} C_VEL
LIN {X 0,Y 299.178,Z 1186.499,A -85,B 0,C 180,E1 21328.551,E2 21328.551} C_VEL
LIN {X 0,Y 299.956,Z 1183.381,A -85,B 0,C 180,E1 21340.195,E2 21340.195} C_VEL
LIN {X 0,Y 307.807,Z 1167.272,A -85,B 0,C 180,E1 21354.761,E2 21354.761} C_VEL
LIN {X 0,Y 328.322,Z 1136.225,A -85,B 0,C 180,E1 21368.308,E2 21368.308} C_VEL
LIN {X 0,Y 358.107,Z 1092.342,A -85,B 0,C 180,E1 21378.858,E2 21378.858} C_VEL
LIN {X 0,Y 391.024,Z 1037.121,A -85,B 0,C 180,E1 21386.499,E2 21386.499} C_VEL
LIN {X 0,Y 421.26,Z 973.018,A -85,B 0,C 180,E1 21391.615,E2 21391.615} C_VEL
LIN {X 0,Y 427.177,Z 954.629,A -85,B 0,C 180,E1 21392.957,E2 21392.957} C_VEL
LIN {X 0,Y 419.087,Z 923.203,A -85,B 0,C 180,E1 21400.999,E2 21400.999} C_VEL
LIN {X 0,Y 411.841,Z 901.842,A -85,B 0,C 180,E1 21410.476,E2 21410.476} C_VEL
LIN {X 0,Y 410.11,Z 895.926,A -85,B 0,C 180,E1 21418.961,E2 21418.961} C_VEL
LIN {X 0,Y 413.375,Z 907.713,A -85,B 0,C 180,E1 21428.999,E2 21428.999} C_VEL
LIN {X 0,Y 421.499,Z 933.382,A -85,B 0,C 180,E1 21438.191,E2 21438.191} C_VEL
LIN {X 0,Y 426.513,Z 960.916,A -85,B 0,C 180,E1 21444.226,E2 21444.226} C_VEL
LIN {X 0,Y 396.928,Z 1029.464,A -85,B 0,C 180,E1 21449.203,E2 21449.203} C_VEL
LIN {X 0,Y 363.758,Z 1089.282,A -85,B 0,C 180,E1 21456.524,E2 21456.524} C_VEL
LIN {X 0,Y 332.598,Z 1138.799,A -85,B 0,C 180,E1 21466.831,E2 21466.831} C_VEL
LIN {X 0,Y 310.28,Z 1175.278,A -85,B 0,C 180,E1 21479.932,E2 21479.932} C_VEL
LIN {X 0,Y 300.793,Z 1196.607,A -85,B 0,C 180,E1 21493.898,E2 21493.898} C_VEL
LIN {X 0,Y 299.112,Z 1204.455,A -85,B 0,C 180,E1 21505.635,E2 21505.635} C_VEL
LIN {X 0,Y 299.213,Z 1203.368,A -85,B 0,C 180,E1 21517.276,E2 21517.276} C_VEL
LIN {X 0,Y 302.759,Z 1191.321,A -85,B 0,C 180,E1 21530.523,E2 21530.523} C_VEL
LIN {X 0,Y 316.606,Z 1164.321,A -85,B 0,C 180,E1 21544.802,E2 21544.802} C_VEL
LIN {X 0,Y 343.253,Z 1122.208,A -85,B 0,C 180,E1 21557.261,E2 21557.261} C_VEL
LIN {X 0,Y 376.452,Z 1067.798,A -85,B 0,C 180,E1 21566.579,E2 21566.579} C_VEL
LIN {X 0,Y 409.356,Z 1003.356,A -85,B 0,C 180,E1 21573.048,E2 21573.048} C_VEL
LIN {X 0,Y 427.38,Z 959.019,A -85,B 0,C 180,E1 21575.872,E2 21575.872} C_VEL
LIN {X 0,Y 420.309,Z 928.586,A -85,B 0,C 180,E1 21583.185,E2 21583.185} C_VEL
LIN {X 0,Y 414.491,Z 910.688,A -85,B 0,C 180,E1 21589.698,E2 21589.698} C_VEL
LIN {X 0,Y 408.909,Z 909.649,A -85,B 0,C 180,E1 21594.59,E2 21594.59} C_VEL
LIN {X 0,Y 407.867,Z 903.461,A -85,B 0,C 180,E1 21601.044,E2 21601.044} C_VEL
LIN {X 0,Y 410.67,Z 915.045,A -85,B 0,C 180,E1 21612.248,E2 21612.248} C_VEL
LIN {X 0,Y 418.115,Z 938.554,A -85,B 0,C 180,E1 21621.218,E2 21621.218} C_VEL
LIN {X 0,Y 422.047,Z 962.495,A -85,B 0,C 180,E1 21626.662,E2 21626.662} C_VEL
LIN {X 0,Y 392.461,Z 1027.093,A -85,B 0,C 180,E1 21631.355,E2 21631.355} C_VEL
LIN {X 0,Y 358.563,Z 1084.078,A -85,B 0,C 180,E1 21638.519,E2 21638.519} C_VEL
LIN {X 0,Y 326.717,Z 1129.78,A -85,B 0,C 180,E1 21648.594,E2 21648.594} C_VEL
LIN {X 0,Y 303.382,Z 1162.701,A -85,B 0,C 180,E1 21661.652,E2 21661.652} C_VEL
LIN {X 0,Y 293.19,Z 1180.439,A -85,B 0,C 180,E1 21675.015,E2 21675.015} C_VEL
LIN {X 0,Y 291.199,Z 1186.746,A -85,B 0,C 180,E1 21688.511,E2 21688.511} C_VEL
LIN {X 0,Y 292.003,Z 1183.631,A -85,B 0,C 180,E1 21700.476,E2 21700.476} C_VEL
LIN {X 0,Y 300.374,Z 1167.53,A -85,B 0,C 180,E1 21715.416,E2 21715.416} C_VEL
LIN {X 0,Y 321.323,Z 1137.306,A -85,B 0,C 180,E1 21728.965,E2 21728.965} C_VEL
LIN {X 0,Y 352.006,Z 1093.797,A -85,B 0,C 180,E1 21739.657,E2 21739.657} C_VEL
LIN {X 0,Y 385.989,Z 1038.61,A -85,B 0,C 180,E1 21747.384,E2 21747.384} C_VEL
LIN {X 0,Y 416.815,Z 975.169,A -85,B 0,C 180,E1 21752.484,E2 21752.484} C_VEL
LIN {X 0,Y 422.38,Z 959.222,A -85,B 0,C 180,E1 21753.62,E2 21753.62} C_VEL
LIN {X 0,Y 415.544,Z 929.781,A -85,B 0,C 180,E1 21761.384,E2 21761.384} C_VEL
LIN {X 0,Y 409.209,Z 909.747,A -85,B 0,C 180,E1 21770.414,E2 21770.414} C_VEL
LIN {X 0,Y 407.536,Z 903.543,A -85,B 0,C 180,E1 21778.955,E2 21778.955} C_VEL
LIN {X 0,Y 410.565,Z 915.574,A -85,B 0,C 180,E1 21789.062,E2 21789.062} C_VEL
LIN {X 0,Y 417.695,Z 940.461,A -85,B 0,C 180,E1 21798.014,E2 21798.014} C_VEL
LIN {X 0,Y 421.515,Z 964.913,A -85,B 0,C 180,E1 21803.442,E2 21803.442} C_VEL
LIN {X 0,Y 390.433,Z 1034.037,A -85,B 0,C 180,E1 21808.605,E2 21808.605} C_VEL
LIN {X 0,Y 355.79,Z 1093.837,A -85,B 0,C 180,E1 21816.245,E2 21816.245} C_VEL
LIN {X 0,Y 324.143,Z 1141.868,A -85,B 0,C 180,E1 21826.773,E2 21826.773} C_VEL
LIN {X 0,Y 302.182,Z 1176.418,A -85,B 0,C 180,E1 21839.874,E2 21839.874} C_VEL
LIN {X 0,Y 292.87,Z 1196.505,A -85,B 0,C 180,E1 21853.596,E2 21853.596} C_VEL
LIN {X 0,Y 291.102,Z 1204.206,A -85,B 0,C 180,E1 21865.515,E2 21865.515} C_VEL
LIN {X 0,Y 291.218,Z 1203.119,A -85,B 0,C 180,E1 21877.477,E2 21877.477} C_VEL
LIN {X 0,Y 295.005,Z 1191.06,A -85,B 0,C 180,E1 21891.087,E2 21891.087} C_VEL
LIN {X 0,Y 309.855,Z 1163.841,A -85,B 0,C 180,E1 21905.773,E2 21905.773} C_VEL
LIN {X 0,Y 337.409,Z 1122.169,A -85,B 0,C 180,E1 21918.257,E2 21918.257} C_VEL
LIN {X 0,Y 370.992,Z 1068.988,A -85,B 0,C 180,E1 21927.455,E2 21927.455} C_VEL
LIN {X 0,Y 404.884,Z 1004.608,A -85,B 0,C 180,E1 21933.961,E2 21933.961} C_VEL
LIN {X 0,Y 422.251,Z 961.597,A -85,B 0,C 180,E1 21936.925,E2 21936.925} C_VEL
LIN {X 0,Y 415.596,Z 931.676,A -85,B 0,C 180,E1 21944.625,E2 21944.625} C_VEL
LIN {X 0,Y 409.287,Z 911.345,A -85,B 0,C 180,E1 21953.591,E2 21953.591} C_VEL
LIN {X 0,Y 408.909,Z 909.649,A -85,B 0,C 180,E1 21954.59,E2 21954.59} C_VEL
LIN {X 0,Y 405.05,Z 912.475,A -85,B 0,C 180,E1 21959.543,E2 21959.543} C_VEL
LIN {X 0,Y 404.935,Z 914.117,A -85,B 0,C 180,E1 21965.355,E2 21965.355} C_VEL
LIN {X 0,Y 409.139,Z 927.185,A -85,B 0,C 180,E1 21974.479,E2 21974.479} C_VEL
LIN {X 0,Y 415.987,Z 953.199,A -85,B 0,C 180,E1 21983.113,E2 21983.113} C_VEL
LIN {X 0,Y 416.973,Z 966.684,A -85,B 0,C 180,E1 21985.876,E2 21985.876} C_VEL
LIN {X 0,Y 386.134,Z 1031.374,A -85,B 0,C 180,E1 21990.724,E2 21990.724} C_VEL
LIN {X 0,Y 351.107,Z 1087.826,A -85,B 0,C 180,E1 21998.081,E2 21998.081} C_VEL
LIN {X 0,Y 318.098,Z 1133.226,A -85,B 0,C 180,E1 22008.591,E2 22008.591} C_VEL
LIN {X 0,Y 294.344,Z 1165.545,A -85,B 0,C 180,E1 22022.378,E2 22022.378} C_VEL
LIN {X 0,Y 284.814,Z 1181.841,A -85,B 0,C 180,E1 22036.14,E2 22036.14} C_VEL
LIN {X 0,Y 283.198,Z 1186.993,A -85,B 0,C 180,E1 22048.469,E2 22048.469} C_VEL
LIN {X 0,Y 284.074,Z 1183.881,A -85,B 0,C 180,E1 22060.772,E2 22060.772} C_VEL
LIN {X 0,Y 292.976,Z 1167.788,A -85,B 0,C 180,E1 22076.106,E2 22076.106} C_VEL
LIN {X 0,Y 314.923,Z 1137.576,A -85,B 0,C 180,E1 22089.913,E2 22089.913} C_VEL
LIN {X 0,Y 346.331,Z 1094.72,A -85,B 0,C 180,E1 22100.579,E2 22100.579} C_VEL
LIN {X 0,Y 381.656,Z 1038.966,A -85,B 0,C 180,E1 22108.414,E2 22108.414} C_VEL
LIN {X 0,Y 413.859,Z 973.95,A -85,B 0,C 180,E1 22113.573,E2 22113.573} C_VEL
LIN {X 0,Y 417.415,Z 962.511,A -85,B 0,C 180,E1 22114.59,E2 22114.59} C_VEL
LIN {X 0,Y 411.414,Z 934.978,A -85,B 0,C 180,E1 22122.203,E2 22122.203} C_VEL
LIN {X 0,Y 405.815,Z 916.336,A -85,B 0,C 180,E1 22131.418,E2 22131.418} C_VEL
LIN {X 0,Y 404.959,Z 911.159,A -85,B 0,C 180,E1 22138.948,E2 22138.948} C_VEL
LIN {X 0,Y 407.574,Z 923.344,A -85,B 0,C 180,E1 22149.129,E2 22149.129} C_VEL
LIN {X 0,Y 414.176,Z 948.787,A -85,B 0,C 180,E1 22158.172,E2 22158.172} C_VEL
LIN {X 0,Y 416.251,Z 969.559,A -85,B 0,C 180,E1 22162.699,E2 22162.699} C_VEL
LIN {X 0,Y 384.27,Z 1037.702,A -85,B 0,C 180,E1 22167.926,E2 22167.926} C_VEL
LIN {X 0,Y 349.385,Z 1095.759,A -85,B 0,C 180,E1 22175.522,E2 22175.522} C_VEL
LIN {X 0,Y 316.331,Z 1143.941,A -85,B 0,C 180,E1 22186.434,E2 22186.434} C_VEL
LIN {X 0,Y 294.083,Z 1177.557,A -85,B 0,C 180,E1 22199.82,E2 22199.82} C_VEL
LIN {X 0,Y 285.035,Z 1196.091,A -85,B 0,C 180,E1 22212.982,E2 22212.982} C_VEL
LIN {X 0,Y 283.091,Z 1203.958,A -85,B 0,C 180,E1 22225.388,E2 22225.388} C_VEL
LIN {X 0,Y 283.227,Z 1202.87,A -85,B 0,C 180,E1 22237.69,E2 22237.69} C_VEL
LIN {X 0,Y 287.082,Z 1191.297,A -85,B 0,C 180,E1 22251.299,E2 22251.299} C_VEL
LIN {X 0,Y 302.373,Z 1164.638,A -85,B 0,C 180,E1 22266.271,E2 22266.271} C_VEL
LIN {X 0,Y 331.071,Z 1122.986,A -85,B 0,C 180,E1 22279.092,E2 22279.092} C_VEL
LIN {X 0,Y 366.59,Z 1068.607,A -85,B 0,C 180,E1 22288.564,E2 22288.564} C_VEL
LIN {X 0,Y 401.32,Z 1004.187,A -85,B 0,C 180,E1 22295.026,E2 22295.026} C_VEL
LIN {X 0,Y 417.531,Z 966.457,A -85,B 0,C 180,E1 22297.538,E2 22297.538} C_VEL
LIN {X 0,Y 411.754,Z 938.08,A -85,B 0,C 180,E1 22305.024,E2 22305.024} C_VEL
LIN {X 0,Y 406.372,Z 918.95,A -85,B 0,C 180,E1 22313.544,E2 22313.544} C_VEL
LIN {X 0,Y 405.05,Z 912.475,A -85,B 0,C 180,E1 22319.543,E2 22319.543} C_VEL
LIN {X 0,Y 402.151,Z 919.357,A -85,B 0,C 180,E1 22322.78,E2 22322.78} C_VEL
LIN {X 0,Y 405.001,Z 931.618,A -85,B 0,C 180,E1 22332.972,E2 22332.972} C_VEL
LIN {X 0,Y 411.153,Z 956.573,A -85,B 0,C 180,E1 22342.004,E2 22342.004} C_VEL
LIN {X 0,Y 411.929,Z 970.874,A -85,B 0,C 180,E1 22345.087,E2 22345.087} C_VEL
LIN {X 0,Y 379.995,Z 1035.264,A -85,B 0,C 180,E1 22350.033,E2 22350.033} C_VEL
LIN {X 0,Y 344.103,Z 1090.946,A -85,B 0,C 180,E1 22357.511,E2 22357.511} C_VEL
LIN {X 0,Y 310.303,Z 1135.614,A -85,B 0,C 180,E1 22368.254,E2 22368.254} C_VEL
LIN {X 0,Y 286.213,Z 1167.094,A -85,B 0,C 180,E1 22382.382,E2 22382.382} C_VEL
LIN {X 0,Y 276.503,Z 1183.244,A -85,B 0,C 180,E1 22397.33,E2 22397.33} C_VEL
LIN {X 0,Y 275.468,Z 1187.219,A -85,B 0,C 180,E1 22411.58,E2 22411.58} C_VEL
LIN {X 0,Y 277.687,Z 1180.843,A -85,B 0,C 180,E1 22425.85,E2 22425.85} C_VEL
LIN {X 0,Y 290.904,Z 1160.359,A -85,B 0,C 180,E1 22441.422,E2 22441.422} C_VEL
LIN {X 0,Y 318.048,Z 1125.509,A -85,B 0,C 180,E1 22454.697,E2 22454.697} C_VEL
LIN {X 0,Y 353.322,Z 1077.571,A -85,B 0,C 180,E1 22464.585,E2 22464.585} C_VEL
LIN {X 0,Y 388.731,Z 1019.177,A -85,B 0,C 180,E1 22471.379,E2 22471.379} C_VEL
LIN {X 0,Y 412.741,Z 968.261,A -85,B 0,C 180,E1 22475.006,E2 22475.006} C_VEL
LIN {X 0,Y 407.385,Z 940.669,A -85,B 0,C 180,E1 22482.911,E2 22482.911} C_VEL
LIN {X 0,Y 402.903,Z 923.906,A -85,B 0,C 180,E1 22491.356,E2 22491.356} C_VEL
LIN {X 0,Y 402.07,Z 918.676,A -85,B 0,C 180,E1 22498.941,E2 22498.941} C_VEL
LIN {X 0,Y 404.549,Z 931.094,A -85,B 0,C 180,E1 22509.197,E2 22509.197} C_VEL
LIN {X 0,Y 410.106,Z 955.899,A -85,B 0,C 180,E1 22518.053,E2 22518.053} C_VEL
LIN {X 0,Y 411.435,Z 973.073,A -85,B 0,C 180,E1 22521.872,E2 22521.872} C_VEL
LIN {X 0,Y 378.029,Z 1041.608,A -85,B 0,C 180,E1 22527.25,E2 22527.25} C_VEL
LIN {X 0,Y 341.52,Z 1099.906,A -85,B 0,C 180,E1 22535.161,E2 22535.161} C_VEL
LIN {X 0,Y 307.773,Z 1147.118,A -85,B 0,C 180,E1 22546.423,E2 22546.423} C_VEL
LIN {X 0,Y 285.355,Z 1179.765,A -85,B 0,C 180,E1 22560.364,E2 22560.364} C_VEL
LIN {X 0,Y 276.252,Z 1198.613,A -85,B 0,C 180,E1 22575.695,E2 22575.695} C_VEL
LIN {X 0,Y 275.423,Z 1204.233,A -85,B 0,C 180,E1 22588.419,E2 22588.419} C_VEL
LIN {X 0,Y 275.621,Z 1200.885,A -85,B 0,C 180,E1 22601.1,E2 22601.1} C_VEL
LIN {X 0,Y 281.568,Z 1186.304,A -85,B 0,C 180,E1 22615.52,E2 22615.52} C_VEL
LIN {X 0,Y 300.194,Z 1157.858,A -85,B 0,C 180,E1 22629.871,E2 22629.871} C_VEL
LIN {X 0,Y 331.426,Z 1114.572,A -85,B 0,C 180,E1 22642.025,E2 22642.025} C_VEL
LIN {X 0,Y 367.741,Z 1059.397,A -85,B 0,C 180,E1 22650.81,E2 22650.81} C_VEL
LIN {X 0,Y 401.63,Z 996.023,A -85,B 0,C 180,E1 22656.639,E2 22656.639} C_VEL
LIN {X 0,Y 412.543,Z 969.833,A -85,B 0,C 180,E1 22658.461,E2 22658.461} C_VEL
LIN {X 0,Y 407.2,Z 941.383,A -85,B 0,C 180,E1 22666.506,E2 22666.506} C_VEL
LIN {X 0,Y 402.673,Z 923.629,A -85,B 0,C 180,E1 22675.654,E2 22675.654} C_VEL
LIN {X 0,Y 402.151,Z 919.357,A -85,B 0,C 180,E1 22682.78,E2 22682.78} C_VEL
LIN {X 0,Y 399.613,Z 930.897,A -85,B 0,C 180,E1 22687.56,E2 22687.56} C_VEL
LIN {X 0,Y 403.779,Z 947.855,A -85,B 0,C 180,E1 22696.726,E2 22696.726} C_VEL
LIN {X 0,Y 407.99,Z 972.703,A -85,B 0,C 180,E1 22704.144,E2 22704.144} C_VEL
LIN {X 0,Y 374.962,Z 1037.369,A -85,B 0,C 180,E1 22709.14,E2 22709.14} C_VEL
LIN {X 0,Y 338.023,Z 1092.81,A -85,B 0,C 180,E1 22716.688,E2 22716.688} C_VEL
LIN {X 0,Y 303.368,Z 1136.941,A -85,B 0,C 180,E1 22727.561,E2 22727.561} C_VEL
LIN {X 0,Y 278.949,Z 1167.359,A -85,B 0,C 180,E1 22741.604,E2 22741.604} C_VEL
LIN {X 0,Y 268.598,Z 1183.495,A -85,B 0,C 180,E1 22756.951,E2 22756.951} C_VEL
LIN {X 0,Y 267.459,Z 1187.466,A -85,B 0,C 180,E1 22771.628,E2 22771.628} C_VEL
LIN {X 0,Y 269.821,Z 1181.167,A -85,B 0,C 180,E1 22786.226,E2 22786.226} C_VEL
LIN {X 0,Y 282.851,Z 1161.996,A -85,B 0,C 180,E1 22801.52,E2 22801.52} C_VEL
LIN {X 0,Y 310.371,Z 1128.139,A -85,B 0,C 180,E1 22815.116,E2 22815.116} C_VEL
LIN {X 0,Y 346.735,Z 1080.616,A -85,B 0,C 180,E1 22825.263,E2 22825.263} C_VEL
LIN {X 0,Y 383.157,Z 1022.732,A -85,B 0,C 180,E1 22832.162,E2 22832.162} C_VEL
LIN {X 0,Y 407.751,Z 971.442,A -85,B 0,C 180,E1 22836.036,E2 22836.036} C_VEL
LIN {X 0,Y 403.17,Z 945.214,A -85,B 0,C 180,E1 22844.061,E2 22844.061} C_VEL
LIN {X 0,Y 399.532,Z 930.406,A -85,B 0,C 180,E1 22852.382,E2 22852.382} C_VEL
LIN {X 0,Y 399.148,Z 926.184,A -85,B 0,C 180,E1 22858.933,E2 22858.933} C_VEL
LIN {X 0,Y 400.981,Z 937.637,A -85,B 0,C 180,E1 22868.731,E2 22868.731} C_VEL
LIN {X 0,Y 405.843,Z 962.053,A -85,B 0,C 180,E1 22877.656,E2 22877.656} C_VEL
LIN {X 0,Y 406.333,Z 977.551,A -85,B 0,C 180,E1 22881.094,E2 22881.094} C_VEL
LIN {X 0,Y 372.442,Z 1044.467,A -85,B 0,C 180,E1 22886.445,E2 22886.445} C_VEL
LIN {X 0,Y 335.57,Z 1101.289,A -85,B 0,C 180,E1 22894.29,E2 22894.29} C_VEL
LIN {X 0,Y 300.764,Z 1148.155,A -85,B 0,C 180,E1 22905.736,E2 22905.736} C_VEL
LIN {X 0,Y 277.543,Z 1180.412,A -85,B 0,C 180,E1 22920.037,E2 22920.037} C_VEL
LIN {X 0,Y 268.341,Z 1198.359,A -85,B 0,C 180,E1 22935.264,E2 22935.264} C_VEL
LIN {X 0,Y 267.408,Z 1203.985,A -85,B 0,C 180,E1 22948.372,E2 22948.372} C_VEL
LIN {X 0,Y 267.67,Z 1200.634,A -85,B 0,C 180,E1 22961.434,E2 22961.434} C_VEL
LIN {X 0,Y 274.061,Z 1186.042,A -85,B 0,C 180,E1 22976.271,E2 22976.271} C_VEL
LIN {X 0,Y 294.237,Z 1157.026,A -85,B 0,C 180,E1 22991.118,E2 22991.118} C_VEL
LIN {X 0,Y 327.645,Z 1112.422,A -85,B 0,C 180,E1 23003.565,E2 23003.565} C_VEL
LIN {X 0,Y 365.873,Z 1055.55,A -85,B 0,C 180,E1 23012.366,E2 23012.366} C_VEL
LIN {X 0,Y 400.606,Z 990.942,A -85,B 0,C 180,E1 23018.036,E2 23018.036} C_VEL
LIN {X 0,Y 407.673,Z 973.879,A -85,B 0,C 180,E1 23019.263,E2 23019.263} C_VEL
LIN {X 0,Y 403.127,Z 946.341,A -85,B 0,C 180,E1 23027.474,E2 23027.474} C_VEL
LIN {X 0,Y 399.4,Z 930.142,A -85,B 0,C 180,E1 23036.71,E2 23036.71} C_VEL
LIN {X 0,Y 399.222,Z 926.857,A -85,B 0,C 180,E1 23042.704,E2 23042.704} C_VEL
LIN {X 0,Y 399.613,Z 930.897,A -85,B 0,C 180,E1 23047.56,E2 23047.56} C_VEL
LIN {X 0,Y 397.935,Z 945.158,A -85,B 0,C 180,E1 23052.249,E2 23052.249} C_VEL
LIN {X 0,Y 402.35,Z 967.884,A -85,B 0,C 180,E1 23060.977,E2 23060.977} C_VEL
LIN {X 0,Y 402.444,Z 978.424,A -85,B 0,C 180,E1 23063.402,E2 23063.402} C_VEL
LIN {X 0,Y 368.019,Z 1042.88,A -85,B 0,C 180,E1 23068.575,E2 23068.575} C_VEL
LIN {X 0,Y 329.689,Z 1097.68,A -85,B 0,C 180,E1 23076.397,E2 23076.397} C_VEL
LIN {X 0,Y 294.469,Z 1140.441,A -85,B 0,C 180,E1 23087.627,E2 23087.627} C_VEL
LIN {X 0,Y 269.894,Z 1169.837,A -85,B 0,C 180,E1 23102.387,E2 23102.387} C_VEL
LIN {X 0,Y 260.292,Z 1184.693,A -85,B 0,C 180,E1 23118.237,E2 23118.237} C_VEL
LIN {X 0,Y 259.45,Z 1187.714,A -85,B 0,C 180,E1 23131.678,E2 23131.678} C_VEL
LIN {X 0,Y 262.314,Z 1180.831,A -85,B 0,C 180,E1 23147.421,E2 23147.421} C_VEL
LIN {X 0,Y 276.934,Z 1160.885,A -85,B 0,C 180,E1 23163.207,E2 23163.207} C_VEL
LIN {X 0,Y 306.56,Z 1126.064,A -85,B 0,C 180,E1 23176.862,E2 23176.862} C_VEL
LIN {X 0,Y 343.921,Z 1078.437,A -85,B 0,C 180,E1 23186.767,E2 23186.767} C_VEL
LIN {X 0,Y 381.243,Z 1019.918,A -85,B 0,C 180,E1 23193.514,E2 23193.514} C_VEL
LIN {X 0,Y 402.996,Z 976.112,A -85,B 0,C 180,E1 23196.729,E2 23196.729} C_VEL
LIN {X 0,Y 399.344,Z 951.952,A -85,B 0,C 180,E1 23204.346,E2 23204.346} C_VEL
LIN {X 0,Y 396.293,Z 937.794,A -85,B 0,C 180,E1 23212.319,E2 23212.319} C_VEL
LIN {X 0,Y 396.067,Z 933.612,A -85,B 0,C 180,E1 23218.925,E2 23218.925} C_VEL
LIN {X 0,Y 397.657,Z 945.234,A -85,B 0,C 180,E1 23228.805,E2 23228.805} C_VEL
LIN {X 0,Y 401.604,Z 969.064,A -85,B 0,C 180,E1 23237.508,E2 23237.508} C_VEL
LIN {X 0,Y 401.373,Z 981.821,A -85,B 0,C 180,E1 23240.276,E2 23240.276} C_VEL
LIN {X 0,Y 366.132,Z 1048.665,A -85,B 0,C 180,E1 23245.755,E2 23245.755} C_VEL
LIN {X 0,Y 327.551,Z 1105.532,A -85,B 0,C 180,E1 23253.922,E2 23253.922} C_VEL
LIN {X 0,Y 291.691,Z 1151.723,A -85,B 0,C 180,E1 23265.944,E2 23265.944} C_VEL
LIN {X 0,Y 268.988,Z 1182.138,A -85,B 0,C 180,E1 23280.438,E2 23280.438} C_VEL
LIN {X 0,Y 260.04,Z 1199.381,A -85,B 0,C 180,E1 23296.507,E2 23296.507} C_VEL
LIN {X 0,Y 259.408,Z 1203.738,A -85,B 0,C 180,E1 23308.322,E2 23308.322} C_VEL
LIN {X 0,Y 259.706,Z 1200.383,A -85,B 0,C 180,E1 23321.79,E2 23321.79} C_VEL
LIN {X 0,Y 266.539,Z 1185.915,A -85,B 0,C 180,E1 23336.969,E2 23336.969} C_VEL
LIN {X 0,Y 287.956,Z 1156.75,A -85,B 0,C 180,E1 23352.218,E2 23352.218} C_VEL
LIN {X 0,Y 321.922,Z 1113.189,A -85,B 0,C 180,E1 23364.552,E2 23364.552} C_VEL
LIN {X 0,Y 360.738,Z 1057.354,A -85,B 0,C 180,E1 23373.289,E2 23373.289} C_VEL
LIN {X 0,Y 395.962,Z 993.931,A -85,B 0,C 180,E1 23378.916,E2 23378.916} C_VEL
LIN {X 0,Y 402.875,Z 978.293,A -85,B 0,C 180,E1 23380.011,E2 23380.011} C_VEL
LIN {X 0,Y 399.227,Z 952.687,A -85,B 0,C 180,E1 23387.907,E2 23387.907} C_VEL
LIN {X 0,Y 396.16,Z 937.495,A -85,B 0,C 180,E1 23396.683,E2 23396.683} C_VEL
LIN {X 0,Y 396.411,Z 933.518,A -85,B 0,C 180,E1 23401.074,E2 23401.074} C_VEL
LIN {X 0,Y 397.398,Z 942.948,A -85,B 0,C 180,E1 23410.986,E2 23410.986} C_VEL
LIN {X 0,Y 397.935,Z 945.158,A -85,B 0,C 180,E1 23412.249,E2 23412.249} C_VEL
LIN {X 0,Y 396.166,Z 962.662,A -85,B 0,C 180,E1 23416.73,E2 23416.73} C_VEL
LIN {X 0,Y 398.04,Z 981.7,A -85,B 0,C 180,E1 23422.507,E2 23422.507} C_VEL
LIN {X 0,Y 362.069,Z 1046.44,A -85,B 0,C 180,E1 23427.803,E2 23427.803} C_VEL
LIN {X 0,Y 322.393,Z 1100.993,A -85,B 0,C 180,E1 23435.836,E2 23435.836} C_VEL
LIN {X 0,Y 286.084,Z 1143.271,A -85,B 0,C 180,E1 23447.482,E2 23447.482} C_VEL
LIN {X 0,Y 261.738,Z 1171.199,A -85,B 0,C 180,E1 23462.389,E2 23462.389} C_VEL
LIN {X 0,Y 252.388,Z 1184.942,A -85,B 0,C 180,E1 23477.863,E2 23477.863} C_VEL
LIN {X 0,Y 251.441,Z 1187.962,A -85,B 0,C 180,E1 23491.732,E2 23491.732} C_VEL
LIN {X 0,Y 254.541,Z 1181.085,A -85,B 0,C 180,E1 23507.971,E2 23507.971} C_VEL
LIN {X 0,Y 270.071,Z 1161.148,A -85,B 0,C 180,E1 23524.165,E2 23524.165} C_VEL
LIN {X 0,Y 300.974,Z 1126.342,A -85,B 0,C 180,E1 23538.009,E2 23538.009} C_VEL
LIN {X 0,Y 340.16,Z 1077.828,A -85,B 0,C 180,E1 23548.067,E2 23548.067} C_VEL
LIN {X 0,Y 378.5,Z 1018.922,A -85,B 0,C 180,E1 23554.725,E2 23554.725} C_VEL
LIN {X 0,Y 398.21,Z 979.807,A -85,B 0,C 180,E1 23557.696,E2 23557.696} C_VEL
LIN {X 0,Y 395.037,Z 956.497,A -85,B 0,C 180,E1 23565.561,E2 23565.561} C_VEL
LIN {X 0,Y 393.037,Z 945.227,A -85,B 0,C 180,E1 23572.255,E2 23572.255} C_VEL
LIN {X 0,Y 392.811,Z 940.975,A -85,B 0,C 180,E1 23578.916,E2 23578.916} C_VEL
LIN {X 0,Y 394.117,Z 952.767,A -85,B 0,C 180,E1 23588.884,E2 23588.884} C_VEL
LIN {X 0,Y 397.253,Z 976.568,A -85,B 0,C 180,E1 23597.534,E2 23597.534} C_VEL
LIN {X 0,Y 396.36,Z 986.108,A -85,B 0,C 180,E1 23599.45,E2 23599.45} C_VEL
LIN {X 0,Y 359.873,Z 1052.5,A -85,B 0,C 180,E1 23605.034,E2 23605.034} C_VEL
LIN {X 0,Y 319.821,Z 1109.176,A -85,B 0,C 180,E1 23613.465,E2 23613.465} C_VEL
LIN {X 0,Y 283.664,Z 1153.94,A -85,B 0,C 180,E1 23625.694,E2 23625.694} C_VEL
LIN {X 0,Y 260.038,Z 1184.403,A -85,B 0,C 180,E1 23641.337,E2 23641.337} C_VEL
LIN {X 0,Y 251.762,Z 1200.115,A -85,B 0,C 180,E1 23657.826,E2 23657.826} C_VEL
LIN {X 0,Y 251.125,Z 1203.485,A -85,B 0,C 180,E1 23671.727,E2 23671.727} C_VEL
LIN {X 0,Y 252.509,Z 1197.872,A -85,B 0,C 180,E1 23685.676,E2 23685.676} C_VEL
LIN {X 0,Y 263.877,Z 1179.329,A -85,B 0,C 180,E1 23702.11,E2 23702.11} C_VEL
LIN {X 0,Y 291.47,Z 1144.782,A -85,B 0,C 180,E1 23717.477,E2 23717.477} C_VEL
LIN {X 0,Y 329.348,Z 1096.872,A -85,B 0,C 180,E1 23728.829,E2 23728.829} C_VEL
LIN {X 0,Y 368.944,Z 1037.91,A -85,B 0,C 180,E1 23736.505,E2 23736.505} C_VEL
LIN {X 0,Y 398.036,Z 981.61,A -85,B 0,C 180,E1 23741.064,E2 23741.064} C_VEL
LIN {X 0,Y 394.806,Z 956.468,A -85,B 0,C 180,E1 23749.455,E2 23749.455} C_VEL
LIN {X 0,Y 392.903,Z 944.865,A -85,B 0,C 180,E1 23756.655,E2 23756.655} C_VEL
LIN {X 0,Y 393.156,Z 940.879,A -85,B 0,C 180,E1 23761.083,E2 23761.083} C_VEL
LIN {X 0,Y 394.137,Z 951.355,A -85,B 0,C 180,E1 23771.606,E2 23771.606} C_VEL
LIN {X 0,Y 396.166,Z 962.662,A -85,B 0,C 180,E1 23776.73,E2 23776.73} C_VEL
LIN {X 0,Y 393.607,Z 982.709,A -85,B 0,C 180,E1 23781.003,E2 23781.003} C_VEL
LIN {X 0,Y 391.684,Z 988.774,A -85,B 0,C 180,E1 23781.84,E2 23781.84} C_VEL
LIN {X 0,Y 355.169,Z 1051.414,A -85,B 0,C 180,E1 23787.155,E2 23787.155} C_VEL
LIN {X 0,Y 315.13,Z 1104.3,A -85,B 0,C 180,E1 23795.246,E2 23795.246} C_VEL
LIN {X 0,Y 278.295,Z 1145.436,A -85,B 0,C 180,E1 23807.07,E2 23807.07} C_VEL
LIN {X 0,Y 253.578,Z 1172.561,A -85,B 0,C 180,E1 23822.392,E2 23822.392} C_VEL
LIN {X 0,Y 244.472,Z 1185.192,A -85,B 0,C 180,E1 23837.464,E2 23837.464} C_VEL
LIN {X 0,Y 243.441,Z 1188.209,A -85,B 0,C 180,E1 23851.788,E2 23851.788} C_VEL
LIN {X 0,Y 246.139,Z 1182.307,A -85,B 0,C 180,E1 23867.222,E2 23867.222} C_VEL
LIN {X 0,Y 262.041,Z 1162.775,A -85,B 0,C 180,E1 23884.355,E2 23884.355} C_VEL
LIN {X 0,Y 293.494,Z 1128.969,A -85,B 0,C 180,E1 23898.528,E2 23898.528} C_VEL
LIN {X 0,Y 332.984,Z 1082.069,A -85,B 0,C 180,E1 23908.645,E2 23908.645} C_VEL
LIN {X 0,Y 372.106,Z 1024.406,A -85,B 0,C 180,E1 23915.42,E2 23915.42} C_VEL
LIN {X 0,Y 393.401,Z 984.1,A -85,B 0,C 180,E1 23918.523,E2 23918.523} C_VEL
LIN {X 0,Y 390.764,Z 960.49,A -85,B 0,C 180,E1 23927.118,E2 23927.118} C_VEL
LIN {X 0,Y 389.12,Z 950.814,A -85,B 0,C 180,E1 23934.427,E2 23934.427} C_VEL
LIN {X 0,Y 389.538,Z 948.319,A -85,B 0,C 180,E1 23938.907,E2 23938.907} C_VEL
LIN {X 0,Y 390.41,Z 960.304,A -85,B 0,C 180,E1 23948.969,E2 23948.969} C_VEL
LIN {X 0,Y 392.842,Z 983.789,A -85,B 0,C 180,E1 23957.476,E2 23957.476} C_VEL
LIN {X 0,Y 391.327,Z 990.48,A -85,B 0,C 180,E1 23958.631,E2 23958.631} C_VEL
LIN {X 0,Y 353.798,Z 1056.099,A -85,B 0,C 180,E1 23964.252,E2 23964.252} C_VEL
LIN {X 0,Y 313.197,Z 1111.476,A -85,B 0,C 180,E1 23972.717,E2 23972.717} C_VEL
LIN {X 0,Y 276.213,Z 1155.411,A -85,B 0,C 180,E1 23985.136,E2 23985.136} C_VEL
LIN {X 0,Y 252.407,Z 1184.586,A -85,B 0,C 180,E1 24000.756,E2 24000.756} C_VEL
LIN {X 0,Y 243.821,Z 1199.863,A -85,B 0,C 180,E1 24017.423,E2 24017.423} C_VEL
LIN {X 0,Y 243.13,Z 1203.238,A -85,B 0,C 180,E1 24031.784,E2 24031.784} C_VEL
LIN {X 0,Y 244.657,Z 1197.619,A -85,B 0,C 180,E1 24046.193,E2 24046.193} C_VEL
LIN {X 0,Y 257.955,Z 1177.674,A -85,B 0,C 180,E1 24063.948,E2 24063.948} C_VEL
LIN {X 0,Y 287.164,Z 1142.939,A -85,B 0,C 180,E1 24079.226,E2 24079.226} C_VEL
LIN {X 0,Y 326.668,Z 1094.479,A -85,B 0,C 180,E1 24090.464,E2 24090.464} C_VEL
LIN {X 0,Y 367.15,Z 1035.209,A -85,B 0,C 180,E1 24097.932,E2 24097.932} C_VEL
LIN {X 0,Y 393.271,Z 986.055,A -85,B 0,C 180,E1 24101.833,E2 24101.833} C_VEL
LIN {X 0,Y 390.724,Z 961.632,A -85,B 0,C 180,E1 24110.474,E2 24110.474} C_VEL
LIN {X 0,Y 389.354,Z 950.233,A -85,B 0,C 180,E1 24118.86,E2 24118.86} C_VEL
LIN {X 0,Y 389.456,Z 949.343,A -85,B 0,C 180,E1 24123.328,E2 24123.328} C_VEL
LIN {X 0,Y 390.88,Z 960.989,A -85,B 0,C 180,E1 24132.878,E2 24132.878} C_VEL
LIN {X 0,Y 393.607,Z 982.709,A -85,B 0,C 180,E1 24141.003,E2 24141.003} C_VEL
LIN {X 0,Y 389.015,Z 991.753,A -85,B 0,C 180,E1 24141.549,E2 24141.549} C_VEL
LIN {X 0,Y 381.511,Z 1002.987,A -85,B 0,C 180,E1 24141.639,E2 24141.639} C_VEL
LIN {X 0,Y 342.215,Z 1064.836,A -85,B 0,C 180,E1 24147.54,E2 24147.54} C_VEL
LIN {X 0,Y 301.246,Z 1115.035,A -85,B 0,C 180,E1 24156.35,E2 24156.35} C_VEL
LIN {X 0,Y 265.454,Z 1152.646,A -85,B 0,C 180,E1 24168.934,E2 24168.934} C_VEL
LIN {X 0,Y 242.376,Z 1177.596,A -85,B 0,C 180,E1 24186.006,E2 24186.006} C_VEL
LIN {X 0,Y 235.809,Z 1187.043,A -85,B 0,C 180,E1 24200.752,E2 24200.752} C_VEL
LIN {X 0,Y 235.344,Z 1187.98,A -85,B 0,C 180,E1 24215.55,E2 24215.55} C_VEL
LIN {X 0,Y 240.876,Z 1179.132,A -85,B 0,C 180,E1 24232.198,E2 24232.198} C_VEL
LIN {X 0,Y 262.603,Z 1155.718,A -85,B 0,C 180,E1 24249.44,E2 24249.44} C_VEL
LIN {X 0,Y 297.975,Z 1118.596,A -85,B 0,C 180,E1 24262.681,E2 24262.681} C_VEL
LIN {X 0,Y 339.785,Z 1067.942,A -85,B 0,C 180,E1 24271.95,E2 24271.95} C_VEL
LIN {X 0,Y 378.524,Z 1008.218,A -85,B 0,C 180,E1 24277.842,E2 24277.842} C_VEL
LIN {X 0,Y 388.621,Z 988.46,A -85,B 0,C 180,E1 24279.335,E2 24279.335} C_VEL
LIN {X 0,Y 386.742,Z 965.79,A -85,B 0,C 180,E1 24288.133,E2 24288.133} C_VEL
LIN {X 0,Y 385.738,Z 956.08,A -85,B 0,C 180,E1 24296.999,E2 24296.999} C_VEL
LIN {X 0,Y 385.829,Z 960.748,A -85,B 0,C 180,E1 24304.74,E2 24304.74} C_VEL
LIN {X 0,Y 387.534,Z 978.802,A -85,B 0,C 180,E1 24313.615,E2 24313.615} C_VEL
LIN {X 0,Y 387.601,Z 992.36,A -85,B 0,C 180,E1 24317.623,E2 24317.623} C_VEL
LIN {X 0,Y 348.849,Z 1058.155,A -85,B 0,C 180,E1 24323.277,E2 24323.277} C_VEL
LIN {X 0,Y 307.513,Z 1112.672,A -85,B 0,C 180,E1 24331.708,E2 24331.708} C_VEL
LIN {X 0,Y 269.603,Z 1155.918,A -85,B 0,C 180,E1 24344.173,E2 24344.173} C_VEL
LIN {X 0,Y 244.105,Z 1185.835,A -85,B 0,C 180,E1 24360.95,E2 24360.95} C_VEL
LIN {X 0,Y 235.886,Z 1199.611,A -85,B 0,C 180,E1 24376.992,E2 24376.992} C_VEL
LIN {X 0,Y 235.134,Z 1202.991,A -85,B 0,C 180,E1 24391.844,E2 24391.844} C_VEL
LIN {X 0,Y 236.802,Z 1197.366,A -85,B 0,C 180,E1 24406.746,E2 24406.746} C_VEL
LIN {X 0,Y 251.035,Z 1177.41,A -85,B 0,C 180,E1 24425.018,E2 24425.018} C_VEL
LIN {X 0,Y 281.798,Z 1142.507,A -85,B 0,C 180,E1 24440.591,E2 24440.591} C_VEL
LIN {X 0,Y 322.185,Z 1094.718,A -85,B 0,C 180,E1 24451.669,E2 24451.669} C_VEL
LIN {X 0,Y 363.699,Z 1035.518,A -85,B 0,C 180,E1 24459.078,E2 24459.078} C_VEL
LIN {X 0,Y 388.459,Z 990.612,A -85,B 0,C 180,E1 24462.588,E2 24462.588} C_VEL
LIN {X 0,Y 386.762,Z 967.971,A -85,B 0,C 180,E1 24470.945,E2 24470.945} C_VEL
LIN {X 0,Y 386.282,Z 955.471,A -85,B 0,C 180,E1 24481.103,E2 24481.103} C_VEL
LIN {X 0,Y 386.679,Z 965.366,A -85,B 0,C 180,E1 24491.295,E2 24491.295} C_VEL
LIN {X 0,Y 388.833,Z 987.308,A -85,B 0,C 180,E1 24500.238,E2 24500.238} C_VEL
LIN {X 0,Y 384.139,Z 998.26,A -85,B 0,C 180,E1 24501.308,E2 24501.308} C_VEL
LIN {X 0,Y 381.511,Z 1002.987,A -85,B 0,C 180,E1 24501.639,E2 24501.639} C_VEL
LIN {X 0,Y 361.798,Z 1031.675,A -85,B 0,C 180,E1 24502.742,E2 24502.742} C_VEL
LIN {X 0,Y 320.72,Z 1087.734,A -85,B 0,C 180,E1 24509.576,E2 24509.576} C_VEL
LIN {X 0,Y 279.756,Z 1132.863,A -85,B 0,C 180,E1 24519.972,E2 24519.972} C_VEL
LIN {X 0,Y 246.099,Z 1166.091,A -85,B 0,C 180,E1 24535.288,E2 24535.288} C_VEL
LIN {X 0,Y 229.842,Z 1183.817,A -85,B 0,C 180,E1 24553.109,E2 24553.109} C_VEL
LIN {X 0,Y 227.279,Z 1188.72,A -85,B 0,C 180,E1 24568.092,E2 24568.092} C_VEL
LIN {X 0,Y 228.705,Z 1185.632,A -85,B 0,C 180,E1 24583.423,E2 24583.423} C_VEL
LIN {X 0,Y 242.455,Z 1169.594,A -85,B 0,C 180,E1 24602.122,E2 24602.122} C_VEL
LIN {X 0,Y 272.374,Z 1140.014,A -85,B 0,C 180,E1 24617.543,E2 24617.543} C_VEL
LIN {X 0,Y 313.569,Z 1096.131,A -85,B 0,C 180,E1 24628.851,E2 24628.851} C_VEL
LIN {X 0,Y 355.942,Z 1040.277,A -85,B 0,C 180,E1 24636.357,E2 24636.357} C_VEL
LIN {X 0,Y 383.849,Z 992.209,A -85,B 0,C 180,E1 24640.385,E2 24640.385} C_VEL
LIN {X 0,Y 382.68,Z 972.485,A -85,B 0,C 180,E1 24648.378,E2 24648.378} C_VEL
LIN {X 0,Y 382.154,Z 963.285,A -85,B 0,C 180,E1 24656.999,E2 24656.999} C_VEL
LIN {X 0,Y 382.088,Z 967.734,A -85,B 0,C 180,E1 24664.58,E2 24664.58} C_VEL
LIN {X 0,Y 383.158,Z 984.875,A -85,B 0,C 180,E1 24673.191,E2 24673.191} C_VEL
LIN {X 0,Y 382.886,Z 996.441,A -85,B 0,C 180,E1 24676.736,E2 24676.736} C_VEL
LIN {X 0,Y 343.002,Z 1061.671,A -85,B 0,C 180,E1 24682.436,E2 24682.436} C_VEL
LIN {X 0,Y 299.462,Z 1116.735,A -85,B 0,C 180,E1 24691.282,E2 24691.282} C_VEL
LIN {X 0,Y 260.749,Z 1158.869,A -85,B 0,C 180,E1 24704.212,E2 24704.212} C_VEL
LIN {X 0,Y 235.784,Z 1186.921,A -85,B 0,C 180,E1 24721.155,E2 24721.155} C_VEL
LIN {X 0,Y 227.957,Z 1199.359,A -85,B 0,C 180,E1 24736.532,E2 24736.532} C_VEL
LIN {X 0,Y 227.124,Z 1202.743,A -85,B 0,C 180,E1 24751.909,E2 24751.909} C_VEL
LIN {X 0,Y 228.973,Z 1197.112,A -85,B 0,C 180,E1 24767.336,E2 24767.336} C_VEL
LIN {X 0,Y 244.18,Z 1177.145,A -85,B 0,C 180,E1 24786.153,E2 24786.153} C_VEL
LIN {X 0,Y 276.646,Z 1142.001,A -85,B 0,C 180,E1 24802.036,E2 24802.036} C_VEL
LIN {X 0,Y 318.433,Z 1094.204,A -85,B 0,C 180,E1 24813.044,E2 24813.044} C_VEL
LIN {X 0,Y 360.784,Z 1035.162,A -85,B 0,C 180,E1 24820.324,E2 24820.324} C_VEL
LIN {X 0,Y 383.716,Z 995.177,A -85,B 0,C 180,E1 24823.36,E2 24823.36} C_VEL
LIN {X 0,Y 382.568,Z 973.136,A -85,B 0,C 180,E1 24831.995,E2 24831.995} C_VEL
LIN {X 0,Y 382.695,Z 962.682,A -85,B 0,C 180,E1 24841.113,E2 24841.113} C_VEL
LIN {X 0,Y 382.744,Z 973.067,A -85,B 0,C 180,E1 24851.645,E2 24851.645} C_VEL
LIN {X 0,Y 384.123,Z 992.904,A -85,B 0,C 180,E1 24859.75,E2 24859.75} C_VEL
LIN {X 0,Y 361.798,Z 1031.675,A -85,B 0,C 180,E1 24862.742,E2 24862.742} C_VEL
LIN {X 0,Y 340.357,Z 1058.5,A -85,B 0,C 180,E1 24864.224,E2 24864.224} C_VEL
LIN {X 0,Y 296.74,Z 1110.385,A -85,B 0,C 180,E1 24872.521,E2 24872.521} C_VEL
LIN {X 0,Y 256.863,Z 1149.794,A -85,B 0,C 180,E1 24884.9,E2 24884.9} C_VEL
LIN {X 0,Y 229.932,Z 1175.423,A -85,B 0,C 180,E1 24901.546,E2 24901.546} C_VEL
LIN {X 0,Y 219.909,Z 1187.54,A -85,B 0,C 180,E1 24920.076,E2 24920.076} C_VEL
LIN {X 0,Y 219.366,Z 1188.477,A -85,B 0,C 180,E1 24935.956,E2 24935.956} C_VEL
LIN {X 0,Y 225.806,Z 1179.64,A -85,B 0,C 180,E1 24953.767,E2 24953.767} C_VEL
LIN {X 0,Y 250.084,Z 1156.235,A -85,B 0,C 180,E1 24971.844,E2 24971.844} C_VEL
LIN {X 0,Y 288.312,Z 1119.159,A -85,B 0,C 180,E1 24985.278,E2 24985.278} C_VEL
LIN {X 0,Y 331.103,Z 1070.313,A -85,B 0,C 180,E1 24994.214,E2 24994.214} C_VEL
LIN {X 0,Y 371.516,Z 1011.137,A -85,B 0,C 180,E1 24999.995,E2 24999.995} C_VEL
LIN {X 0,Y 379.173,Z 996.468,A -85,B 0,C 180,E1 25001.313,E2 25001.313} C_VEL
LIN {X 0,Y 378.539,Z 977.454,A -85,B 0,C 180,E1 25009.629,E2 25009.629} C_VEL
LIN {X 0,Y 378.585,Z 969.817,A -85,B 0,C 180,E1 25018.875,E2 25018.875} C_VEL
LIN {X 0,Y 378.466,Z 981.362,A -85,B 0,C 180,E1 25028.673,E2 25028.673} C_VEL
LIN {X 0,Y 378.206,Z 1000.583,A -85,B 0,C 180,E1 25035.834,E2 25035.834} C_VEL
LIN {X 0,Y 336.842,Z 1065.436,A -85,B 0,C 180,E1 25041.617,E2 25041.617} C_VEL
LIN {X 0,Y 292.422,Z 1119.412,A -85,B 0,C 180,E1 25050.564,E2 25050.564} C_VEL
LIN {X 0,Y 252.128,Z 1161.385,A -85,B 0,C 180,E1 25064.115,E2 25064.115} C_VEL
LIN {X 0,Y 226.929,Z 1188.684,A -85,B 0,C 180,E1 25082.105,E2 25082.105} C_VEL
LIN {X 0,Y 219.329,Z 1200.863,A -85,B 0,C 180,E1 25100.042,E2 25100.042} C_VEL
LIN {X 0,Y 219.129,Z 1202.496,A -85,B 0,C 180,E1 25111.979,E2 25111.979} C_VEL
LIN {X 0,Y 221.163,Z 1196.859,A -85,B 0,C 180,E1 25127.969,E2 25127.969} C_VEL
LIN {X 0,Y 237.414,Z 1176.879,A -85,B 0,C 180,E1 25147.356,E2 25147.356} C_VEL
LIN {X 0,Y 271.416,Z 1141.796,A -85,B 0,C 180,E1 25163.43,E2 25163.43} C_VEL
LIN {X 0,Y 314.741,Z 1093.908,A -85,B 0,C 180,E1 25174.397,E2 25174.397} C_VEL
LIN {X 0,Y 358.263,Z 1034.517,A -85,B 0,C 180,E1 25181.606,E2 25181.606} C_VEL
LIN {X 0,Y 379.018,Z 999.321,A -85,B 0,C 180,E1 25184.293,E2 25184.293} C_VEL
LIN {X 0,Y 378.481,Z 979.237,A -85,B 0,C 180,E1 25192.585,E2 25192.585} C_VEL
LIN {X 0,Y 378.91,Z 969.777,A -85,B 0,C 180,E1 25201.124,E2 25201.124} C_VEL
LIN {X 0,Y 378.635,Z 979.31,A -85,B 0,C 180,E1 25211.117,E2 25211.117} C_VEL
LIN {X 0,Y 378.878,Z 998.498,A -85,B 0,C 180,E1 25218.998,E2 25218.998} C_VEL
LIN {X 0,Y 340.357,Z 1058.5,A -85,B 0,C 180,E1 25224.224,E2 25224.224} C_VEL
LIN {X 0,Y 317.422,Z 1083.208,A -85,B 0,C 180,E1 25226.17,E2 25226.17} C_VEL
LIN {X 0,Y 272.745,Z 1130.326,A -85,B 0,C 180,E1 25236.277,E2 25236.277} C_VEL
LIN {X 0,Y 236.142,Z 1163.58,A -85,B 0,C 180,E1 25250.877,E2 25250.877} C_VEL
LIN {X 0,Y 215.682,Z 1182.944,A -85,B 0,C 180,E1 25269.421,E2 25269.421} C_VEL
LIN {X 0,Y 211.271,Z 1189.215,A -85,B 0,C 180,E1 25287.947,E2 25287.947} C_VEL
LIN {X 0,Y 213.004,Z 1186.132,A -85,B 0,C 180,E1 25304.434,E2 25304.434} C_VEL
LIN {X 0,Y 228.642,Z 1170.109,A -85,B 0,C 180,E1 25324.322,E2 25324.322} C_VEL
LIN {X 0,Y 262.868,Z 1139.322,A -85,B 0,C 180,E1 25340.686,E2 25340.686} C_VEL
LIN {X 0,Y 307.106,Z 1094.752,A -85,B 0,C 180,E1 25351.832,E2 25351.832} C_VEL
LIN {X 0,Y 351.295,Z 1038.695,A -85,B 0,C 180,E1 25358.999,E2 25358.999} C_VEL
LIN {X 0,Y 374.411,Z 1001.023,A -85,B 0,C 180,E1 25362.154,E2 25362.154} C_VEL
LIN {X 0,Y 374.424,Z 982.929,A -85,B 0,C 180,E1 25370.693,E2 25370.693} C_VEL
LIN {X 0,Y 374.686,Z 976.838,A -85,B 0,C 180,E1 25378.863,E2 25378.863} C_VEL
LIN {X 0,Y 374.177,Z 987.445,A -85,B 0,C 180,E1 25388.186,E2 25388.186} C_VEL
LIN {X 0,Y 373.308,Z 1004.94,A -85,B 0,C 180,E1 25394.953,E2 25394.953} C_VEL
LIN {X 0,Y 331.013,Z 1068.781,A -85,B 0,C 180,E1 25400.725,E2 25400.725} C_VEL
LIN {X 0,Y 285.492,Z 1122.022,A -85,B 0,C 180,E1 25409.794,E2 25409.794} C_VEL
LIN {X 0,Y 244.22,Z 1163.2,A -85,B 0,C 180,E1 25423.683,E2 25423.683} C_VEL
LIN {X 0,Y 219.525,Z 1188.463,A -85,B 0,C 180,E1 25441.121,E2 25441.121} C_VEL
LIN {X 0,Y 211.352,Z 1200.612,A -85,B 0,C 180,E1 25459.662,E2 25459.662} C_VEL
LIN {X 0,Y 211.117,Z 1202.249,A -85,B 0,C 180,E1 25472.054,E2 25472.054} C_VEL
LIN {X 0,Y 213.382,Z 1196.606,A -85,B 0,C 180,E1 25488.647,E2 25488.647} C_VEL
LIN {X 0,Y 230.749,Z 1176.615,A -85,B 0,C 180,E1 25508.63,E2 25508.63} C_VEL
LIN {X 0,Y 266.467,Z 1141.521,A -85,B 0,C 180,E1 25524.89,E2 25524.89} C_VEL
LIN {X 0,Y 311.578,Z 1093.183,A -85,B 0,C 180,E1 25535.86,E2 25535.86} C_VEL
LIN {X 0,Y 356.043,Z 1033.707,A -85,B 0,C 180,E1 25542.916,E2 25542.916} C_VEL
LIN {X 0,Y 374.262,Z 1003.04,A -85,B 0,C 180,E1 25545.37,E2 25545.37} C_VEL
LIN {X 0,Y 374.341,Z 983.789,A -85,B 0,C 180,E1 25554.158,E2 25554.158} C_VEL
LIN {X 0,Y 375.01,Z 976.802,A -85,B 0,C 180,E1 25561.136,E2 25561.136} C_VEL
LIN {X 0,Y 374.438,Z 986.504,A -85,B 0,C 180,E1 25571.243,E2 25571.243} C_VEL
LIN {X 0,Y 374.08,Z 1002.737,A -85,B 0,C 180,E1 25578.093,E2 25578.093} C_VEL
LIN {X 0,Y 332.969,Z 1064.02,A -85,B 0,C 180,E1 25583.573,E2 25583.573} C_VEL
LIN {X 0,Y 317.422,Z 1083.208,A -85,B 0,C 180,E1 25586.17,E2 25586.17} C_VEL
LIN {X 0,Y 293.393,Z 1105.685,A -85,B 0,C 180,E1 25588.682,E2 25588.682} C_VEL
LIN {X 0,Y 249.711,Z 1146.756,A -85,B 0,C 180,E1 25600.617,E2 25600.617} C_VEL
LIN {X 0,Y 216.848,Z 1174.912,A -85,B 0,C 180,E1 25618.37,E2 25618.37} C_VEL
LIN {X 0,Y 205.087,Z 1186.442,A -85,B 0,C 180,E1 25635.005,E2 25635.005} C_VEL
LIN {X 0,Y 203.433,Z 1189.446,A -85,B 0,C 180,E1 25652.14,E2 25652.14} C_VEL
LIN {X 0,Y 208.029,Z 1183.118,A -85,B 0,C 180,E1 25671.381,E2 25671.381} C_VEL
LIN {X 0,Y 230.538,Z 1163.061,A -85,B 0,C 180,E1 25690.847,E2 25690.847} C_VEL
LIN {X 0,Y 270.114,Z 1128.273,A -85,B 0,C 180,E1 25705.745,E2 25705.745} C_VEL
